    // Application specific
    Mover : REFERENCE TO FB_Mover;
END_VAR
VAR_OUTPUT
    (* standart Ausgänge *)
    xOUT_ErrFlag  : BOOL;            // Error Flag 
    xOUT_Busy     : BOOL;            // Baustein befindet sich im Ablauf 
    xOUT_Done     : BOOL;            // Baustein hat den Ablauf beendet 		
    xOUT_Ready    : BOOL;            // Ready to begin: should be the same state as done	
    xOUT_Timeout  : BOOL;            // Timeout FB 
    xOUT_InitDone : BOOL;            // initialisierung fertig
    xOUT_Wait     : BOOL;            // Wartet auf Bedingung
    iOUT_Step     : ST140_Measure_e; // Aktueller Schritt 
    sOUT_Step     : STRING;          // Aktueller Schritt but in string format
    bOUT_Error    : BYTE;            // Fehlernummer

    iOUT_ProcessCompletion : INT;  //process completion: express in % (0-100)
    xOUT_MoverFree         : BOOL; // The mover is free to move

END_VAR
VAR
    (* Standard *)
    (* Schritt *)
    iLastStep : ST140_Measure_e; // Merker letzter Schritt 
    iPreStep  : ST140_Measure_e; // Schritt zurück nach Alarm 
    iAktStep  : ST140_Measure_e; // aktueller Schritt

    // Trigger Starten 
    rtSTART : R_TRIG;
    // Timer TimeOut 
    TON_Timeout : TON;

    (* Bausteine *)
    arr_rMeasureTrack_Right : ARRAY[0..1] OF ARRAY[0..MEASURE_PER_PIECE - 1] OF REAL;
    arr_rMeasureTrack_Left  : ARRAY[0..1] OF ARRAY[0..MEASURE_PER_PIECE - 1] OF REAL;

    i            : INT;
    measureIndex : INT; // measure index

    testLevel_Min_Left_NOK  : BOOL; // TRUE when powder level is under the minimum
    testLevel_Max_Left_NOK  : BOOL; // TRUE when powder level is above the maximum
    testLevel_Min_Right_NOK : BOOL; // TRUE when powder level is under the minimum
    testLevel_Max_Right_NOK : BOOL; // TRUE when powder level is above the maximum

    visu_shuttle_x_position : LREAL; // position of the shuttle used in visu
	
	divisor_height_correction : LREAL := 4; // this divisor is used to reduce oscillation during height correction
	// because we may not fix the height on the very next shuttle

END_VAR
VAR CONSTANT
    MEASURE_SIMULATION : BOOL := FALSE; // Set to TRUE to simulate this part of the program
    MEASURE_PER_PIECE  : INT  := 3;     // this must be greater than 1 !
END_VAR

(*******************************************************************)
(* Trigger  *)
(*******************************************************************)
(* Zurücksetzen *)
IF xIN_RESET THEN
    iPreStep  := ST140_Measure_e.RESET;
    iOUT_Step := ST140_Measure_e.RESET;
END_IF;

(* Error Quittieren *)
IF (bOUT_Error <> 0) AND xIN_Quit THEN
    xOUT_ErrFlag := FALSE;
    bOUT_Error   := 0;
    iOUT_Step    := iPreStep; // iPreStep;
END_IF;

(*******************************************************************)
(* Timer *)
(*******************************************************************)
TON_Timeout(IN := xIN_NextStep AND (iLastStep = iOUT_Step) (*todo FG *) ,
            PT := tIN_Timeout);

(*******************************************************************)
(* Bausteine *)
(*******************************************************************)

(*******************************************************************)
(* OUTPUTS *)
(*******************************************************************)
// Error Flag
xOUT_ErrFlag := (bOUT_Error <> 0) OR (ST140_Measure_e.ERROR = iOUT_Step);
// Baustein befindet sich im Ablauf 
xOUT_Busy := (iOUT_Step > ST140_Measure_e.READY) AND (iOUT_Step < ST140_Measure_e.DONE);
// Baustein hat den Ablauf beendet
xOUT_Done := (iOUT_Step = ST140_Measure_e.DONE);
// Process ready
xOUT_Ready := (iOUT_Step = ST140_Measure_e.READY);
// Timeout FB 				 		
xOUT_Timeout := TON_Timeout.Q;
// Itialisierung fertig			
xOUT_InitDone := (iOUT_Step = ST140_Measure_e.READY) OR
                 (iOUT_Step = ST140_Measure_e.DONE);

// Aktueller Schritt			
iOUT_Step := iOUT_Step; //Im Ablauf gesetzt		
sOUT_Step := TO_STRING(iOUT_Step);
//Fehlernummer	 
bOUT_Error := bOUT_Error; //Im Ablauf/FB gesetzt	
(* Warte (alle Schritte wo auf FG oder Teile gewartet wird) *)
xOUT_Wait := (iOUT_Step = ST140_Measure_e.DONE) OR
             (iOUT_Step = ST140_Measure_e.READY) OR
             (iOUT_Step = ST140_Measure_e.START) OR
             (iOUT_Step = ST140_Measure_e.waitOnMover) OR
             (iOUT_Step = ST140_Measure_e.SYNC_MOVER_LEAVE);

xOUT_MoverFree :=
    NOT (iOUT_Step >= ST140_Measure_e.MOVER_NEEDED_OP AND iOUT_Step < ST140_Measure_e.MOVER_FREE_OP) AND
    (iOUT_Step >= ST140_Measure_e.READY) AND
    (iOUT_Step < ST140_Measure_e.ERROR);

iOUT_ProcessCompletion := F_GetPercent_2(iOUT_Step,
                                         ST140_Measure_e.waitOnMover,
                                         ST140_Measure_e.DONE,
                                         ST140_Measure_e.waitOnMover,
                                         ST140_Measure_e.DONE);

(*******************************************************************)
(* Ablauf *)
(*******************************************************************)

(* Sperren *)
IF xIN_Sperre THEN
    iPreStep  := ST140_Measure_e.RESET;
    iOUT_Step := ST140_Measure_e.RESET;
    RETURN;
END_IF;

(* Schritt Merker *)
IF iAktStep <> iOUT_Step THEN
    iLastStep := iAktStep;
    iAktStep  := iOUT_Step;
END_IF

(* START *)
rtSTART(CLK := xIN_Start);

IF __ISVALIDREF(Mover) THEN
    visu_shuttle_x_position := Mover.MovingProcessOffset;
ELSE
    visu_shuttle_x_position := 0.0;
END_IF

IF 0 = bOUT_Error THEN
    // put error conditions here
ELSIF iOUT_Step < ST140_Measure_e.ERROR THEN
    iOUT_Step := ST140_Measure_e.ERROR;
END_IF

(*******************************************************************)
(* Schrittkette  *)
(*******************************************************************)
CASE iOUT_Step OF

(***** RESET *****)
ST140_Measure_e.RESET: (* Schritt 0-99 *)
    //Initialisierungen
    //Start Init Ablauf
    IF xIN_Init THEN
        iOUT_Step := ST140_Measure_e.INIT;
        //Start Manu Ablauf
    ELSIF enIN_State = StateMANU AND xIN_NextStep THEN
        iOUT_Step := ST140_Measure_e.INIT;
    END_IF;

(***** INIT *****)
ST140_Measure_e.INIT: (* Grundstellung ? *)
    IF MEASURE_PER_PIECE < 2 THEN
        bOUT_Error := 4;
    END_IF

    iOUT_Step := ST140_Measure_e.READY;

(***** READY / INIT DONE *****)
ST140_Measure_e.READY: (* Start AUTO:END:LEER:STEP *)
    IF xIN_Start THEN  //IF rtSTART.Q THEN
        iOUT_Step := ST140_Measure_e.START;
    END_IF

(***** START  ZYKLISCH *****)
ST140_Measure_e.START: (*  *)
    IF xIN_NextStep AND pxFG_Freigabe^ THEN
        iOUT_Step := ST140_Measure_e.waitOnMover;
        iPreStep  := ST140_Measure_e.waitOnMover;
    END_IF;

ST140_Measure_e.waitOnMover:
    IF xIN_NextStep AND __ISVALIDREF(Mover) OR HMI.bArForceCyclusState[StationList_e.ST140] THEN
        IF Mover.GetLastStationDone() >= INT#140 THEN
            iOUT_Step := ST140_Measure_e.SYNC_MOVER_LEAVE;
        ELSIF Mover.GetLastStationDone() < INT#130 THEN
            iOUT_Step := ST140_Measure_e.SYNC_MOVER_LEAVE;
        ELSE
            MEMSET(ADR(arr_rMeasureTrack_Right), 0, SIZEOF(arr_rMeasureTrack_Right));
            MEMSET(ADR(arr_rMeasureTrack_Left), 0, SIZEOF(arr_rMeasureTrack_Left));

            measureIndex := 0;
            iOUT_Step    := ST140_Measure_e.Measure_right;
        END_IF
    END_IF

ST140_Measure_e.Measure_right:
    IF xIN_NextStep AND TRUE THEN
        arr_rMeasureTrack_Right[LaserPlace_e.NearTrack][measureIndex] :=
            UINT_TO_REAL(IN.AI01_ST140_level_track_side) * 0.001;

        arr_rMeasureTrack_Right[LaserPlace_e.NearDoor][measureIndex] :=
            UINT_TO_REAL(IN.AI02_ST140_level_door_side) * 0.001;

        measureIndex := measureIndex + 1;

        IF measureIndex >= MEASURE_PER_PIECE THEN
            IF _20_AUTO.recipe.st140.xIsTypeMiniOrSmart THEN
                iOUT_Step := ST140_Measure_e.Move_shuttle_to_pos_left;
            ELSE
                iOUT_Step := ST140_Measure_e.Save_result_in_mover;
            END_IF

            iOUT_Step := ST140_Measure_e.Move_shuttle_to_pos_left;
        ELSE
            iOUT_Step := ST140_Measure_e.Move_shuttle_relative_right;
        END_IF
    END_IF

ST140_Measure_e.Move_shuttle_relative_right:
    IF __ISVALIDREF(Mover) THEN
        IF Mover.MoveRelativeInsideStation(20.0 / (MEASURE_PER_PIECE - 1)) THEN
            iOUT_Step := ST140_Measure_e.Measure_right;
            iPreStep  := ST140_Measure_e.Measure_right;
        END_IF
    ELSE
        bOUT_Error := 10;
    END_IF

ST140_Measure_e.Move_shuttle_to_pos_left:
    IF __ISVALIDREF(Mover) THEN
        IF _20_AUTO.recipe.st140.xIsTypeMiniOrSmart THEN
            IF Mover.MoveRelativeInsideStation(100.0) THEN
                iOUT_Step    := ST140_Measure_e.Measure_left;
                iPreStep     := ST140_Measure_e.Measure_left;
                measureIndex := 0;
            END_IF
        ELSE
            iOUT_Step := ST140_Measure_e.Save_result_in_mover;
            iPreStep  := ST140_Measure_e.Save_result_in_mover;
        END_IF
    ELSE
        bOUT_Error := 11;
    END_IF

ST140_Measure_e.Measure_left:
    IF xIN_NextStep AND __ISVALIDREF(Mover) AND_THEN Mover.IsInStationPos() THEN
        arr_rMeasureTrack_Left[LaserPlace_e.NearTrack][measureIndex] :=
            UINT_TO_REAL(IN.AI01_ST140_level_track_side) * 0.001;

        arr_rMeasureTrack_Left[LaserPlace_e.NearDoor][measureIndex] :=
            UINT_TO_REAL(IN.AI02_ST140_level_door_side) * 0.001;

        measureIndex := measureIndex + 1;

        IF measureIndex >= MEASURE_PER_PIECE THEN
            iOUT_Step := ST140_Measure_e.Save_result_in_mover;
            iPreStep  := ST140_Measure_e.Save_result_in_mover;
        ELSE
            iOUT_Step := ST140_Measure_e.Move_shuttle_relative_left;
        END_IF
    END_IF

ST140_Measure_e.Move_shuttle_relative_left:
    IF __ISVALIDREF(Mover) THEN
        IF Mover.MoveRelativeInsideStation(20.0 / (MEASURE_PER_PIECE - 1)) THEN
            iOUT_Step := ST140_Measure_e.Measure_left;
            iPreStep  := ST140_Measure_e.Measure_left;
        END_IF
    ELSE
        bOUT_Error := 12;
    END_IF

ST140_Measure_e.Save_result_in_mover:

    testLevel_Min_Left_NOK  := FALSE;
    testLevel_Max_Left_NOK  := FALSE;
    testLevel_Min_Right_NOK := FALSE;
    testLevel_Max_Right_NOK := FALSE;

    IF NOT (MEASURE_SIMULATION AND CONST.USE_SIMULATION) THEN

        FOR i := 0 TO MEASURE_PER_PIECE - 1 BY 1 DO
            IF arr_rMeasureTrack_Right[LaserPlace_e.NearTrack][i] < _20_AUTO.recipe.st140.rMinHeightSensorRight OR
               arr_rMeasureTrack_Right[LaserPlace_e.NearDoor][i] < _20_AUTO.recipe.st140.rMinHeightSensorRight THEN
                // min value of the sensor means maximum fill
                testLevel_Max_Right_NOK := TRUE;
            END_IF

            IF arr_rMeasureTrack_Right[LaserPlace_e.NearTrack][i] > _20_AUTO.recipe.st140.rMaxHeightSensorRight OR
               arr_rMeasureTrack_Right[LaserPlace_e.NearDoor][i] > _20_AUTO.recipe.st140.rMaxHeightSensorRight THEN
                // max value of the sensor means minimum fill
                testLevel_Min_Right_NOK := TRUE;
            END_IF
        END_FOR

        IF _20_AUTO.recipe.st140.xIsTypeMiniOrSmart THEN
            FOR i := 0 TO MEASURE_PER_PIECE - 1 BY 1 DO
                IF arr_rMeasureTrack_Left[LaserPlace_e.NearTrack][i] < _20_AUTO.recipe.st140.rMinHeightSensorLeft OR
                   arr_rMeasureTrack_Left[LaserPlace_e.NearDoor][i] < _20_AUTO.recipe.st140.rMinHeightSensorLeft THEN
                    // min value of the sensor means maximum fill
                    testLevel_Max_Left_NOK := TRUE;
                END_IF

                IF arr_rMeasureTrack_Left[LaserPlace_e.NearTrack][i] > _20_AUTO.recipe.st140.rMaxHeightSensorLeft OR
                   arr_rMeasureTrack_Left[LaserPlace_e.NearDoor][i] > _20_AUTO.recipe.st140.rMaxHeightSensorLeft THEN
                    // max value of the sensor means minimum fill
                    testLevel_Min_Left_NOK := TRUE;
                END_IF
            END_FOR
        END_IF

    END_IF

    IF testLevel_Min_Left_NOK OR testLevel_Max_Left_NOK OR testLevel_Min_Right_NOK OR testLevel_Max_Right_NOK THEN
        IF __ISVALIDREF(Mover) THEN
            IF NOT Mover.SetLastStation(-140) THEN
                ASSERT(0);
            END_IF

            // All minimum
            IF (testLevel_Min_Left_NOK AND testLevel_Min_Right_NOK) THEN
                Mover.SetErrorCode(CONCAT(INT_TO_STRING(Mover.GetLastStationDone()), '-D All min'));

                // All maximum
            ELSIF (testLevel_Max_Left_NOK AND testLevel_Max_Right_NOK) THEN
                Mover.SetErrorCode(CONCAT(INT_TO_STRING(Mover.GetLastStationDone()), '-E All max'));

                // Both in error
            ELSIF (testLevel_Min_Left_NOK OR testLevel_Max_Left_NOK) AND
                  (testLevel_Min_Right_NOK OR testLevel_Max_Right_NOK) THEN
                Mover.SetErrorCode(CONCAT(INT_TO_STRING(Mover.GetLastStationDone()), '-F Both left and right'));

                // min and max error on left
            ELSIF (testLevel_Min_Left_NOK AND testLevel_Max_Left_NOK) THEN
                Mover.SetErrorCode(CONCAT(INT_TO_STRING(Mover.GetLastStationDone()), '-G Both left'));

                // min and max error on right
            ELSIF (testLevel_Min_Right_NOK AND testLevel_Max_Right_NOK) THEN
                Mover.SetErrorCode(CONCAT(INT_TO_STRING(Mover.GetLastStationDone()), '-H Both right'));

            ELSIF testLevel_Min_Left_NOK THEN
                Mover.SetErrorCode(CONCAT(INT_TO_STRING(Mover.GetLastStationDone()), '-I Min left'));

            ELSIF testLevel_Max_Left_NOK THEN
                Mover.SetErrorCode(CONCAT(INT_TO_STRING(Mover.GetLastStationDone()), '-J Max left'));

            ELSIF testLevel_Min_Right_NOK THEN
                Mover.SetErrorCode(CONCAT(INT_TO_STRING(Mover.GetLastStationDone()), '-K Min right'));

            ELSIF testLevel_Max_Right_NOK THEN
                Mover.SetErrorCode(CONCAT(INT_TO_STRING(Mover.GetLastStationDone()), '-L Min right'));

            ELSE
                ASSERT(0); // Oops ... read the condition again !
            END_IF
        END_IF

    ELSE
        IF __ISVALIDREF(Mover) THEN
            IF NOT Mover.SetLastStation(140) THEN
                ASSERT(0);
            END_IF
        END_IF
    END_IF

	// Adding a value makes the axis go down
	// Substracting a value makes the axis go up
    IF __ISVALIDREF(Mover) AND_THEN Mover.GetLastStationDone() = 130 THEN
        IF testLevel_Min_Left_NOK THEN
            GVL.ST130_01Y_Feedback_Offset := GVL.ST130_01Y_Feedback_Offset - 0.1;
        END_IF
        IF testLevel_Max_Left_NOK THEN
            GVL.ST130_01Y_Feedback_Offset := GVL.ST130_01Y_Feedback_Offset + 0.1;
        END_IF
        IF testLevel_Min_Right_NOK THEN
            GVL.ST130_01Y_Feedback_Offset := GVL.ST130_01Y_Feedback_Offset - 0.1;
        END_IF
        IF testLevel_Max_Right_NOK THEN
            GVL.ST130_01Y_Feedback_Offset := GVL.ST130_01Y_Feedback_Offset + 0.1;
        END_IF
    END_IF

	// Adding a value makes the axis go down
	// Substracting a value makes the axis go up
    IF __ISVALIDREF(Mover) AND_THEN Mover.GetLastStationDone() = 135 THEN
        IF testLevel_Min_Left_NOK THEN
            GVL.ST135_01Y_Feedback_Offset := GVL.ST135_01Y_Feedback_Offset - 0.1;
        END_IF
        IF testLevel_Max_Left_NOK THEN
            GVL.ST135_01Y_Feedback_Offset := GVL.ST135_01Y_Feedback_Offset + 0.1;
        END_IF
        IF testLevel_Min_Right_NOK THEN
            GVL.ST135_01Y_Feedback_Offset := GVL.ST135_01Y_Feedback_Offset - 0.1;
        END_IF
        IF testLevel_Max_Right_NOK THEN
            GVL.ST135_01Y_Feedback_Offset := GVL.ST135_01Y_Feedback_Offset + 0.1;
        END_IF
    END_IF

    iOUT_Step := ST140_Measure_e.SYNC_MOVER_LEAVE;

ST140_Measure_e.SYNC_MOVER_LEAVE:
    // The mover needs to be taken by MoverMan
    IF NOT __ISVALIDREF(Mover) THEN
        iOUT_Step := ST140_Measure_e.DONE;
    END_IF

(***** DONE *****)
ST140_Measure_e.DONE: (* Letzter Schritt  *)
    IF NOT xIN_AlarmAktiv THEN
        //AUTO
        IF (enIN_State = StateAUTO) AND xIN_RestartCYCL THEN
            iOUT_Step := ST140_Measure_e.START;
            //STEP / END / LEERFAHREN restart
        ELSIF (enIN_State < StateAUTO) AND (enIN_State >= enState.StateSTEP) AND xIN_RestartCYCL THEN
            iOUT_Step := ST140_Measure_e.START;
            //STEP / END / LEERFAHREN fertig
        ELSIF (enIN_State = StateREADY) THEN
            iOUT_Step := ST140_Measure_e.READY;
        END_IF;
    END_IF;

(************ ERROR *************)
ST140_Measure_e.ERROR: (* ERROR *) ;

END_CASE;

END_FUNCTION_BLOCK

// ---- POUs/20_AUTO/ST145/FB_AUT_145.TcPOU
FUNCTION_BLOCK FB_AUT_145 EXTENDS FB_AUT_ABSTRACT
(****************************************************************************)
(*	POU_AUT_zxx			Bausteinaufrufe Station	zxx							*)
(*	Status				ungetestet											*)
(*  Version:			1.0													*)
(*	Beschrieb:																*)
(*																			*)
(*	Abläufe:			FB_ABLzxxA		Hauptablauf							*)
(*																			*)
(*																			*)
(* 	25.09.2019/Dj															*)
(****************************************************************************)
(*	dd.mm.yyyy   KZ    x.y			Beschrieb								*)
(****************************************************************************)
VAR_INPUT
    (* spezifische Eingänge *)

END_VAR
VAR_OUTPUT
    (* spezifische Ausgänge *)

END_VAR
VAR
    (* Bausteine *)
    fb_Pnp    : FB_ABL_145_Pnp;
    fb_Feeder : FB_ABL_145_Feeder;

    fb_stat_pnp    : FB_AUT_Statistics;
    fb_stat_Feeder : FB_AUT_Statistics;

END_VAR

VAR CONSTANT
    ROT_TABLE_FREE_MAX_Y : REAL := 200.0; // If Y and Z axis is more than this value, the feeder cannot move
    ROT_TABLE_FREE_MAX_Z : REAL := 200.0; // If Z and Y axis is more than this value, the feeder cannot move

    PNP_VERTICAL_MAX_Z : REAL := 50.0; // If Z axis is more than this value, the horizontal axis of the pnp cannot move
END_VAR

(*******************************************************************)
(* Timer *)
(*******************************************************************)

(*******************************************************************)
(* Flanken / Merker *)
(*******************************************************************)
//MANU CYCLE
IF (enIN_State = StateMANU) AND xIN_ManuCycle THEN
    xManuCycle := TRUE;
END_IF;

IF (enIN_State <> StateMANU) OR xOUT_Done THEN
    xManuCycle := FALSE;
END_IF

//NEXT STEP
xNextStep := (enIN_State > StateSTEP) OR
             ((enIN_State = StateSTEP) AND xIN_Step) OR
             ((enIN_State = StateMANU) AND xManuCycle);

//RESET
xReset := (enIN_State < StateREADY) AND (enIN_State <> StateINIT) AND NOT xManuCycle;

(*******************************************************************)
(* Bausteinaufrufe Abläufe *)
(*******************************************************************)

xRelease := MAIN.MoverMan.IsProcessUsed(THIS^);

fb_Pnp(xIN_Reset          := xReset,
       xIN_Init           := xIN_Init,
       xIN_Quit           := xIN_Quit,
       xIN_Start          := enIN_State >= enState.StateLEER AND xRelease,
       xIN_Sperre         := NOT xIN_On,
       xIN_NextStep       := xNextStep,
       xIN_AlarmAktiv     := xIN_AlarmAktiv,
       xIN_DryCycle       := xIN_DryCycle,
       xIN_RestartCYCL    := enIN_State >= enState.StateLEER,
       enIN_State         := enIN_State,
       tIN_Timeout        := tIN_Timeout,
       pxFG_Freigabe      := ADR(xRelease),
       Mover              := THIS^.Mover,
       xIN_PceReadyToPick := fb_Feeder.xOUT_Done,
       xIN_HorAxisFree    := ST145_Axis.axis145_02Z.rActPos < ROT_TABLE_FREE_MAX_Y);

fb_Feeder(xIN_Reset       := xReset,
          xIN_Init        := xIN_Init,
          xIN_Quit        := xIN_Quit,
          xIN_Start       := enIN_State >= enState.StateLEER AND xRelease,
          xIN_Sperre      := NOT xIN_On,
          xIN_NextStep    := xNextStep,
          xIN_AlarmAktiv  := xIN_AlarmAktiv,
          xIN_DryCycle    := xIN_DryCycle,
          xIN_RestartCYCL := enIN_State >= enState.StateLEER,
          enIN_State      := enIN_State,
          tIN_Timeout     := tIN_Timeout,
          pxFG_Freigabe   := ADR(xRelease),
          // special
          xIN_PickPiece            := fb_Pnp.xOUT_PickPiece,
          xIN_RotTableBlockedByPnp := (ST145_Axis.axis145_01Y.rActPos > ROT_TABLE_FREE_MAX_Y) AND
                                      (ST145_Axis.axis145_02Z.rActPos > ROT_TABLE_FREE_MAX_Z));

fb_stat_pnp(xIN_Enable  := enState.StateAUTO = enIN_State,
            xIN_Waiting := fb_Pnp.xOUT_Wait,
            xIN_Running := (fb_Pnp.iOUT_Step >= ST145_Pnp_e.START) AND
                           (fb_Pnp.iOUT_Step <= ST145_Pnp_e.DONE),
            // Since we use a mover system, a cycle is done when we are waiting on a mover
            xIN_Done := fb_Pnp.iOUT_Step = ST145_Pnp_e.waitOnMover);

fb_stat_Feeder(xIN_Enable  := enState.StateAUTO = enIN_State,
               xIN_Waiting := fb_feeder.xOUT_Wait,
               xIN_Running := (fb_feeder.iOUT_Step >= ST145_Feeder_e.START) AND
                              (fb_feeder.iOUT_Step <= ST145_Feeder_e.DONE),
               xIN_Done := fb_feeder.iOUT_Step = ST145_Feeder_e.DONE);

(*******************************************************************)
(* Mover reset flags *)
(*******************************************************************)

(*******************************************************************)
(* OUTPUT *)
(*******************************************************************)
xOUT_InitDone := fb_Pnp.xOUT_InitDone AND fb_Feeder.xOUT_InitDone;
xOUT_Ready    := fb_Pnp.xOUT_Ready AND fb_Feeder.xOUT_Ready;
xOUT_Done     := fb_Pnp.xOUT_Done; // we ignore feeder
xOUT_ErrFlag  := fb_Pnp.xOUT_ErrFlag OR fb_Feeder.xOUT_ErrFlag;
xOUT_Wait     := fb_Pnp.xOUT_Wait AND fb_Feeder.xOUT_Wait;
xOUT_AlarmST  := xOUT_ErrFlag;

(*******************************************************************)
(* Bausteinaufruf Error Station *)
(*******************************************************************)
// POU_ERR_VORLAGE(xIN_QUIT:=xIN_Quit , pstrArIN_ALARM:=ADR(HMI.strArALARM[1]));

(* % of completion of the process *)
PROPERTY iCompletionPC : INT
GET
iCompletionPC := THIS^.fb_Pnp.iOUT_ProcessCompletion;
END_GET
END_PROPERTY

PROPERTY ProcessExecution : ProcessExecution_e
GET
ProcessExecution := THIS^._ProcessExecution;
END_GET
SET
THIS^._ProcessExecution := ProcessExecution;
END_SET
END_PROPERTY

PROPERTY xBusy : BOOL
GET
xBusy := THIS^.fb_Pnp.xOUT_Busy;
END_GET
SET
END_SET
END_PROPERTY

PROPERTY xDone : BOOL
GET
xDone := THIS^.fb_Pnp.xOUT_Ready OR THIS^.fb_Pnp.xOUT_Done;
END_GET
END_PROPERTY

PROPERTY xMoverPathFree : BOOL
GET
xMoverPathFree := THIS^.fb_Pnp.xOUT_MoverFree OR THIS^.fb_Pnp.xOUT_Ready OR THIS^.fb_Pnp.xOUT_Done;
END_GET
END_PROPERTY

PROPERTY xMoverShouldLeave : BOOL
GET
xMoverShouldLeave := THIS^.fb_Pnp.iOUT_Step = ST145_Pnp_e.SYNC_MOVER_LEAVE;
END_GET
END_PROPERTY

END_FUNCTION_BLOCK

// ---- POUs/20_AUTO/ST145/FB_ABL_145_Pnp.TcPOU
FUNCTION_BLOCK FB_ABL_145_Pnp
(****************************************************************************************)
(*	TITEL				laden kristall- Modul	    										*)
(*	Status				ungetestet                         								*)
(*	Beschrieb:			Ablaufbeschreibung												*)
(*																						*)
(*	Steps:	self-explained using enum													*)
(***********************************Revisionen*******************************************)
(*	see github blames																	*)
(****************************************************************************************)

VAR_INPUT
    xIN_Reset       : BOOL;          // Schrittkette zurücksetzen 
    xIN_Init        : BOOL;          // Initialisieren
    xIN_Quit        : BOOL;          // Fehler quittieren 
    xIN_Start       : BOOL;          // Startbefehl
    xIN_Sperre      : BOOL;          // FB Sperren 
    xIN_NextStep    : BOOL;          // Nächsten Schritt ausführen 
    xIN_AlarmAktiv  : BOOL;          // Anlage hat Alarm
    xIN_DryCycle    : BOOL;          // Fahren ohne Teile
    xIN_RestartCYCL : BOOL;          // Zyklus erneut starten im STEP, END, LEERFAHREN
    enIN_State      : enState;       // Status Anlage
    tIN_Timeout     : TIME := T#10s; // Timout

    pxFG_Freigabe : POINTER TO BOOL; //Freigabe von Station

    // Application specific
    Mover              : REFERENCE TO FB_Mover;
    xIN_PceReadyToPick : BOOL; // the piece(s) is/are ready to picked
    xIN_HorAxisFree    : BOOL; // TRUE when the vertical is up enough
END_VAR
VAR_OUTPUT
    (* standart Ausgänge *)
    xOUT_ErrFlag  : BOOL;        // Error Flag 
    xOUT_Busy     : BOOL;        // Baustein befindet sich im Ablauf 
    xOUT_Done     : BOOL;        // Baustein hat den Ablauf beendet 		
    xOUT_Ready    : BOOL;        // Ready to begin, should be the same state as done	
    xOUT_Timeout  : BOOL;        // Timeout FB 
    xOUT_InitDone : BOOL;        // initialisierung fertig
    xOUT_Wait     : BOOL;        // Wartet auf Bedingung
    iOUT_Step     : ST145_Pnp_e; // Aktueller Schritt 
    sOUT_Step     : STRING;      // Aktueller Schritt but in string format
    bOUT_Error    : BYTE;        // Fehlernummer

    iOUT_ProcessCompletion : INT;  //process completion, express in % (0-100)
    xOUT_MoverFree         : BOOL; // The mover is free to move
    xOUT_PickPiece         : BOOL; // Set to true when a piece is picked

END_VAR
VAR
    (* Standard *)
    (* Schritt *)
    iLastStep : ST145_Pnp_e; // Merker letzter Schritt 
    iPreStep  : ST145_Pnp_e; // Schritt zurück nach Alarm 
    iAktStep  : ST145_Pnp_e; // aktueller Schritt

    // Trigger Starten 
    rtSTART : R_TRIG;
    // Timer TimeOut 
    TON_Timeout : TON;

    (* Bausteine *)

    (* Spezial *)
    fb_axis145_01Y : FB_AxisLM_V1_1;
    fb_axis145_02Z : FB_AxisLM_V1_1;

    fb_PnpHorAxis : FB_LinearMotionMan;
    fb_PnpVerAxis : FB_LinearMotionMan;

    fb_simu_axis145_01Y : FB_Simu_AxisLM_V1_1;
    fb_simu_axis145_02Z : FB_Simu_AxisLM_V1_1;

    fb_vakumGriperLeft    : FB_ZylMo2El_V2_1;
    fb_vakumGriperRight   : FB_ZylMo2El_V2_1;
    simu_vacumGriperLeft  : FB_Simu_Zyl2Pos;
    simu_vacumGriperRight : FB_Simu_Zyl2Pos;

END_VAR
VAR CONSTANT
    PNP_SIMULATION : BOOL := FALSE; // Set to TRUE to simulate this part of the program
END_VAR

(*******************************************************************)
(* Trigger  *)
(*******************************************************************)
(* Zurücksetzen *)
IF xIN_RESET THEN
    iPreStep  := ST145_Pnp_e.RESET;
    iOUT_Step := ST145_Pnp_e.RESET;
END_IF;

(* Error Quittieren *)
IF (bOUT_Error <> 0) AND xIN_Quit THEN
    xOUT_ErrFlag := FALSE;
    bOUT_Error   := 0;
    iOUT_Step    := iPreStep;
END_IF;

(*******************************************************************)
(* Timer *)
(*******************************************************************)
TON_Timeout(IN := xIN_NextStep AND (iLastStep = iOUT_Step) (*todo FG *) ,
            PT := tIN_Timeout);

(*******************************************************************)
(* Bausteine *)
(*******************************************************************)
fb_PnpHorAxis(config          := _20_AUTO.recipe.linearAxis[LinearAxis_e.ST145_01Y],
              xIN_Init        := enIN_State = enState.StateINIT,
              xIN_Reset       := xIN_Reset,
              lrIN_CurrPos    := fb_axis145_01Y.rOUT_ActPos,
              lrIN_Delta_mm   := 0.5,
              iIN_CurrentStep := iOUT_Step,
              iIN_moveNumber  := ST145_PnpHorPos_e._max);

fb_simu_axis145_01Y(xIN_Enable          := PNP_SIMULATION AND CONST.USE_SIMULATION,
                    bIN_AxisCntr        := fb_axis145_01Y.bOUT_AxisCntr,
                    wIN_AxisState       := ST145_Axis.axis145_01Y.wState,
                    udiIN_HomingTime_ms := 2000,
                    pIN_axisSimu        := ADR(SIMU.axis_ref[Axis_e.ST145_01Y]),
                    pIN_axisHW          := ADR(ST145_Axis.axis145_01Y.axis),
                    rIN_PosActual       := fb_axis145_01Y.rOUT_ActPos,
                    rIN_PosMax          := ST145_Axis.const145_01Y.POS_MAX,
                    rIN_PosMin          := ST145_Axis.const145_01Y.POS_MIN,
                    rIN_PixMax          := 100,
                    rIN_PixMin          := 0);

fb_axis145_01Y(enIN_State       := enIN_State,
               parIN_Buttons    := ADR(AXIS.btTeachArAxis[Axis_e.ST145_01Y]),
               xIN_DisButtons   :=,
               xIN_Quit         := xIN_Quit,
               xIN_PARAMok      := TRUE, (*TODO*)
               xIN_FREE         := TRUE,
               xIN_FREE_HOME    := TRUE,
               rIN_POSMIN       := ST145_Axis.const145_01Y.POS_MIN,
               rIN_POSMAX       := ST145_Axis.const145_01Y.POS_MAX,
               rIN_VELOMAX      := ST145_Axis.const145_01Y.VELO_MAX,
               rIN_VELOMANU     := ST145_Axis.const145_01Y.VELO_MANU,
               rIN_VELOOPEN     := ST145_Axis.const145_01Y.VELO_MANU / 4,
               rIN_JogInc       := AXIS.rTeachIncAxis,
               xIN_Execute      := fb_PnpHorAxis.xOUT_Execute,
               xIN_Home         := ST145_Pnp_e.Init_HomeHorizontals = iAktStep,
               xIN_Relative     :=,
               rIN_Position     := TO_REAL(fb_PnpHorAxis.OUT_MoveProfile.lrPosition),
               rIN_Velocity     := TO_REAL(fb_PnpHorAxis.OUT_MoveProfile.lrVelocity),
               rIN_Acceleration := TO_REAL(fb_PnpHorAxis.OUT_MoveProfile.lrAccel),
               rIN_Deceleration := TO_REAL(fb_PnpHorAxis.OUT_MoveProfile.lrDecel),
               rIN_Jerk         := TO_REAL(fb_PnpHorAxis.OUT_MoveProfile.lrJerk),
               rIN_PosManu      :=
               TO_REAL(_20_AUTO.recipe
                           .linearAxis[LinearAxis_e.ST145_01Y].movesList[AXIS.bTeachPos[Axis_e.ST145_01Y]].lrPosition),
               rIN_VeloJogManu := TO_REAL(Axis.rJogVelo_pc),
               xIN_Reset       := (ST145_Pnp_e.RESET = iAktStep) OR xIN_Reset,
               // The simu fb gives the hardware state when we are not in simu
               wAxisState    := fb_simu_axis145_01Y.wOUT_AxisState,
               rOUT_ActPos   => st145_axis.axis145_01Y.rActPos,
               bOUT_AxisCntr => ST145_Axis.axis145_01Y.bCtrlHi,
               axisIN_REF    := fb_simu_axis145_01Y.pOUT_axisRef^);

fb_PnpVerAxis(config          := _20_AUTO.recipe.linearAxis[LinearAxis_e.ST145_02Z],
              xIN_Init        := enIN_State = enState.StateINIT,
              xIN_Reset       := xIN_Reset,
              lrIN_CurrPos    := fb_axis145_02Z.rOUT_ActPos,
              lrIN_Delta_mm   := 1.0,
              iIN_CurrentStep := iOUT_Step,
              iIN_moveNumber  := ST145_PnpVerPos_e._max);

fb_simu_axis145_02Z(xIN_Enable          := PNP_SIMULATION AND CONST.USE_SIMULATION,
                    bIN_AxisCntr        := fb_axis145_02Z.bOUT_AxisCntr,
                    wIN_AxisState       := ST145_Axis.axis145_02Z.wState,
                    udiIN_HomingTime_ms := 2000,
                    pIN_axisSimu        := ADR(SIMU.axis_ref[Axis_e.ST145_02Z]),
                    pIN_axisHW          := ADR(ST145_Axis.axis145_02Z.axis),
                    rIN_PosActual       := fb_axis145_02Z.rOUT_ActPos,
                    rIN_PosMax          := ST145_Axis.const145_02Z.POS_MAX,
                    rIN_PosMin          := ST145_Axis.const145_02Z.POS_MIN,
                    rIN_PixMax          := 100,
                    rIN_PixMin          := 0);

fb_axis145_02Z(enIN_State       := enIN_State,
               parIN_Buttons    := ADR(AXIS.btTeachArAxis[Axis_e.ST145_02Z]),
               xIN_DisButtons   :=,
               xIN_Quit         := xIN_Quit,
               xIN_PARAMok      := TRUE, (*TODO*)
               xIN_FREE         := TRUE,
               xIN_FREE_HOME    := TRUE,
               rIN_POSMIN       := ST145_Axis.const145_02Z.POS_MIN,
               rIN_POSMAX       := ST145_Axis.const145_02Z.POS_MAX,
               rIN_VELOMAX      := ST145_Axis.const145_02Z.VELO_MAX,
               rIN_VELOMANU     := ST145_Axis.const145_02Z.VELO_MANU,
               rIN_VELOOPEN     := ST145_Axis.const145_02Z.VELO_MANU / 4,
               rIN_JogInc       := AXIS.rTeachIncAxis,
               xIN_Execute      := fb_PnpVerAxis.xOUT_Execute,
               xIN_Home         := ST145_Pnp_e.Init_HomeVerticals = iAktStep,
               xIN_Relative     :=,
               rIN_Position     := TO_REAL(fb_PnpVerAxis.OUT_MoveProfile.lrPosition),
               rIN_Velocity     := TO_REAL(fb_PnpVerAxis.OUT_MoveProfile.lrVelocity),
               rIN_Acceleration := TO_REAL(fb_PnpVerAxis.OUT_MoveProfile.lrAccel),
               rIN_Deceleration := TO_REAL(fb_PnpVerAxis.OUT_MoveProfile.lrDecel),
               rIN_Jerk         := TO_REAL(fb_PnpVerAxis.OUT_MoveProfile.lrJerk),
               rIN_PosManu      :=
               TO_REAL(_20_AUTO.recipe
                           .linearAxis[LinearAxis_e.ST145_02Z].movesList[AXIS.bTeachPos[Axis_e.ST145_02Z]].lrPosition),
               rIN_VeloJogManu := TO_REAL(Axis.rJogVelo_pc),
               xIN_Reset       := (ST145_Pnp_e.RESET = iAktStep) OR xIN_Reset,
               // The simu fb gives the hardware state when we are not in simu
               wAxisState    := fb_simu_axis145_02Z.wOUT_AxisState,
               rOUT_ActPos   => st145_axis.axis145_02Z.rActPos,
               bOUT_AxisCntr => ST145_Axis.axis145_02Z.bCtrlHi,
               axisIN_REF    := fb_simu_axis145_02Z.pOUT_axisRef^);

//////////////////////////////////
fb_vakumGriperLeft(xIN_Reset    := xIN_Reset OR (ST145_Pnp_e.RESET = iOUT_Step),
                   xIN_Quit     := xIN_Quit,
                   xIN_Manu     := enState.StateMANU = enIN_State,
                   pbtIN_Button := ADR(HMI.btManuCylinders[StationList_e.ST145][1]),
                   xIN_GS       := simu_vacumGriperLeft.xOUT_inGS,
                   xIN_AS       := simu_vacumGriperLeft.xOUT_inAS,
                   xIN_FREE     := TRUE,
                   xINtoGS      := ST145_Pnp_e.Vacum_off = iOUT_Step,
                   xINtoAS      := _20_AUTO.recipe.st145.xUseVerLeft AND ST145_Pnp_e.Vacum_on = iOUT_Step,
                   tIN_ErrAS    := DINT_TO_TIME(_20_AUTO.recipe.cylinder2Pos[StationList_e.ST145]
                                                    [ST145_Cylinders_e.VakuumgreiferLinks].toAS_alarm_time),
                   tIN_ErrGS := DINT_TO_TIME(_20_AUTO.recipe.cylinder2Pos[StationList_e.ST145]
                                                 [ST145_Cylinders_e.VakuumgreiferLinks].toGS_alarm_time),
                   tIN_WaitAS := DINT_TO_TIME(_20_AUTO.recipe.cylinder2Pos[StationList_e.ST145]
                                                  [ST145_Cylinders_e.VakuumgreiferLinks].toAS_wait_time),
                   tIN_WaitGS := DINT_TO_TIME(_20_AUTO.recipe.cylinder2Pos[StationList_e.ST145]
                                                  [ST145_Cylinders_e.VakuumgreiferLinks].toGS_wait_time));

simu_vacumGriperLeft(xIN_Enable := PNP_SIMULATION AND CONST.USE_SIMULATION,
                     xIN_inGS   := NOT IO_BOX.I1600_ST145_vakum_teil_in_greiffer_left,
                     xIN_inAS   := IO_BOX.I1600_ST145_vakum_teil_in_greiffer_left,
                     xIN_valve  := fb_vakumGriperLeft.xOUT_VALVE,
                     tIN_GS_ms  := 0,    //ms
                     tIN_AS_ms  := 200); //ms

fb_vakumGriperRight(xIN_Reset    := xIN_Reset OR (ST145_Pnp_e.RESET = iOUT_Step),
                    xIN_Quit     := xIN_Quit,
                    xIN_Manu     := enState.StateMANU = enIN_State,
                    pbtIN_Button := ADR(HMI.btManuCylinders[StationList_e.ST145][2]),
                    xIN_GS       := simu_vacumGriperRight.xOUT_inGS,
                    xIN_AS       := simu_vacumGriperRight.xOUT_inAS,
                    xIN_FREE     := TRUE,
                    xINtoGS      := ST145_Pnp_e.Vacum_off = iOUT_Step,
                    xINtoAS      := _20_AUTO.recipe.st145.xUseVerRight AND ST145_Pnp_e.Vacum_on = iOUT_Step,
                    tIN_ErrAS    := DINT_TO_TIME(_20_AUTO.recipe.cylinder2Pos[StationList_e.ST145]
                                                     [ST145_Cylinders_e.VakuumgreiferRechts].toAS_alarm_time),
                    tIN_ErrGS := DINT_TO_TIME(_20_AUTO.recipe.cylinder2Pos[StationList_e.ST145]
                                                  [ST145_Cylinders_e.VakuumgreiferRechts].toGS_alarm_time),
                    tIN_WaitAS := DINT_TO_TIME(_20_AUTO.recipe.cylinder2Pos[StationList_e.ST145]
                                                   [ST145_Cylinders_e.VakuumgreiferRechts].toAS_wait_time),
                    tIN_WaitGS := DINT_TO_TIME(_20_AUTO.recipe.cylinder2Pos[StationList_e.ST145]
                                                   [ST145_Cylinders_e.VakuumgreiferRechts].toGS_wait_time));

simu_vacumGriperRight(xIN_Enable := PNP_SIMULATION AND CONST.USE_SIMULATION,
                      xIN_inGS   := NOT IO_BOX.I1601_ST145_vakum_teil_in_greiffer_right,
                      xIN_inAS   := IO_BOX.I1601_ST145_vakum_teil_in_greiffer_right,
                      xIN_valve  := fb_vakumGriperRight.xOUT_VALVE,
                      tIN_GS_ms  := 0,    //ms
                      tIN_AS_ms  := 200); //ms

(*******************************************************************)
(* OUTPUTS *)
(*******************************************************************)
// Error Flag 
xOUT_ErrFlag := (bOUT_Error <> 0) OR (ST145_Pnp_e.ERROR = iOUT_Step);
// Baustein befindet sich im Ablauf 
xOUT_Busy := (iOUT_Step > ST145_Pnp_e.READY) AND (iOUT_Step < ST145_Pnp_e.DONE);
// Baustein hat den Ablauf beendet
xOUT_Done := (iOUT_Step = ST145_Pnp_e.DONE);
// Process ready
xOUT_Ready := (iOUT_Step = ST145_Pnp_e.READY) OR (iOUT_Step = ST145_Pnp_e.waitOnMover);
// Timeout FB 				 		
xOUT_Timeout := TON_Timeout.Q;
// Itialisierung fertig			
xOUT_InitDone := (iOUT_Step = ST145_Pnp_e.READY) OR (iOUT_Step = ST145_Pnp_e.waitOnMover);
// Aktueller Schritt			
iOUT_Step := iOUT_Step; //Im Ablauf gesetzt		
sOUT_Step := TO_STRING(iOUT_Step);
//Fehlernummer	 
bOUT_Error := bOUT_Error; //Im Ablauf/FB gesetzt	
(* Warte (alle Schritte wo auf FG oder Teile gewartet wird) *)
xOUT_Wait := (iOUT_Step = ST145_Pnp_e.DONE) OR
             (iOUT_Step = ST145_Pnp_e.READY) OR
             (iOUT_Step = ST145_Pnp_e.START) OR
             (iOUT_Step = ST145_Pnp_e.waitOnMover) OR
             (iOUT_Step = ST145_Pnp_e.SYNC_MOVER_LEAVE) OR
             (iOUT_Step = ST145_Pnp_e.PnP_WaitOnFeeder);

xOUT_MoverFree := iOUT_Step >= ST145_Pnp_e.MOVER_FREE_OP AND iOUT_Step < ST145_Pnp_e.MOVER_NEEDED_OP;

iOUT_ProcessCompletion := F_GetPercent_2(iAktStep,
                                         ST145_Pnp_e.Pnp_Hor_ToRotTablePos,
                                         ST145_Pnp_e.Pnp_Hor_ToTrackPos,
                                         ST145_Pnp_e.Pnp_Ver_ShuttleDown,
                                         ST145_Pnp_e.SYNC_MOVER_LEAVE);

xOUT_PickPiece := iOUT_Step = ST145_Pnp_e.Vacum_on; // the feeder needs to move only when 
// the pnp is outside the feeder

// TODO Valve should not be set when we are in simulation !
IO_BOX.Q0200_14_ST145_vakum_greifer_links :=
    fb_vakumGriperLeft.xOUT_VALVE AND NOT (PNP_SIMULATION AND CONST.USE_SIMULATION);

IO_BOX.Q0201_14_ST145_vakum_greifer_rechts :=
    fb_vakumGriperRight.xOUT_VALVE AND NOT (PNP_SIMULATION AND CONST.USE_SIMULATION);

(*******************************************************************)
(* Ablauf *)
(*******************************************************************)

(* Sperren *)
IF xIN_Sperre THEN
    iPreStep  := ST145_Pnp_e.RESET;
    iOUT_Step := ST145_Pnp_e.RESET;
    RETURN;
END_IF;

(* Schritt Merker *)
IF iAktStep <> iOUT_Step THEN
    iLastStep := iAktStep;
    iAktStep  := iOUT_Step;
END_IF

(* START *)
rtSTART(CLK := xIN_Start);

IF 0 = bOUT_Error THEN
    IF fb_axis145_01Y.xOUT_ErrFlag THEN
        bOUT_Error := 11;
    ELSIF fb_axis145_02Z.xOUT_ErrFlag THEN
        bOUT_Error := 12;
    ELSIF fb_vakumGriperLeft.xOUT_ErrFlag THEN
        bOUT_Error := 13;
    ELSIF fb_vakumGriperRight.xOUT_ErrFlag THEN
        bOUT_Error := 14;
    END_IF
ELSIF iOUT_Step < ST145_Pnp_e.ERROR THEN
    iPreStep  := ST145_Pnp_e.INIT;
    iOUT_Step := ST145_Pnp_e.ERROR;
END_IF

(*******************************************************************)
(* Schrittkette  *)
(*******************************************************************)
CASE iOUT_Step OF

(***** RESET *****)
ST145_Pnp_e.RESET: (* Schritt 0-99 *)
    //Initialisierungen
    //Start Init Ablauf
    IF xIN_Init THEN
        iOUT_Step := ST145_Pnp_e.INIT;
        //Start Manu Ablauf
    ELSIF enIN_State = StateMANU AND xIN_NextStep THEN
        iOUT_Step := ST145_Pnp_e.INIT;
    END_IF;

(***** INIT *****)
ST145_Pnp_e.INIT: (* Grundstellung ? *)
    IF fb_axis145_02Z.xOUT_HOMED THEN
        iOUT_Step := ST145_Pnp_e.Init_VerticalsUp;
    ELSE
        iOUT_Step := ST145_Pnp_e.Init_HomeVerticals;
    END_IF;

ST145_Pnp_e.Init_HomeVerticals:
    IF fb_axis145_02Z.xOUT_HOMED THEN
        iOUT_Step := ST145_Pnp_e.Init_VerticalsUp;
    END_IF

ST145_Pnp_e.Init_VerticalsUp:
    IF fb_vakumGriperLeft.xIN_AS OR fb_vakumGriperRight.xIN_AS THEN
        IF fb_PnpVerAxis.MoveTo(ST145_PnpVerPos_e.UpFull).xOUT_InPos THEN
            IF fb_axis145_01Y.xOUT_HOMED THEN
                iOUT_Step := ST145_Pnp_e.Init_HorizontalsToTrack;
            ELSE
                iOUT_Step := ST145_Pnp_e.Init_HomeHorizontals;
            END_IF
        END_IF
    ELSE
        IF fb_PnpVerAxis.MoveTo(ST145_PnpVerPos_e.UpEmpty).xOUT_InPos THEN
            IF fb_axis145_01Y.xOUT_HOMED THEN
                iOUT_Step := ST145_Pnp_e.Init_HorizontalsToTrack;
            ELSE
                iOUT_Step := ST145_Pnp_e.Init_HomeHorizontals;
            END_IF
        END_IF
    END_IF

ST145_Pnp_e.Init_HomeHorizontals:
    IF fb_axis145_01Y.xOUT_HOMED THEN
        iOUT_Step := ST145_Pnp_e.Init_HorizontalsToTrack;
    END_IF

ST145_Pnp_e.Init_HorizontalsToTrack:
    fb_axis145_02Z.rIN_Velocity := ST145_Axis.const145_02Z.VELO_MANU;

    IF fb_PnpHorAxis.MoveTo(ST145_PnpHorPos_e.GS_Before_placement).xOUT_InPos THEN
        iOUT_Step := ST145_Pnp_e.Init_check_if_pces_handled;
    END_IF

ST145_Pnp_e.Init_check_if_pces_handled:
    IF (NOT _20_AUTO.recipe.st145.xUseVerLeft AND fb_vakumGriperLeft.xOUT_inAS) OR
       (NOT _20_AUTO.recipe.st145.xUseVerRight AND fb_vakumGriperRight.xOUT_inAS) THEN
        // ERROR: a piece is present in an unused gripper
        bOUT_Error := 1;
        iOUT_Step  := ST145_Pnp_e.ERROR;

    ELSIF _20_AUTO.recipe.st145.xUseVerLeft AND
          NOT fb_vakumGriperLeft.xOUT_inAS AND
          _20_AUTO.recipe.st145.xUseVerRight AND
          fb_vakumGriperRight.xOUT_inAS THEN
        // ERROR:  Initialisation failed. A piece is missing in the left griper.
        bOUT_Error := 2;
        iOUT_Step  := ST145_Pnp_e.ERROR;

    ELSIF _20_AUTO.recipe.st145.xUseVerLeft AND
          fb_vakumGriperLeft.xOUT_inAS AND
          _20_AUTO.recipe.st145.xUseVerRight AND
          NOT fb_vakumGriperRight.xOUT_inAS THEN
        // ERROR:  Initialisation failed. A piece is missing in the right griper.
        bOUT_Error := 3;
        iOUT_Step  := ST145_Pnp_e.ERROR;

    ELSIF NOT fb_vakumGriperLeft.xOUT_inAS AND NOT fb_vakumGriperRight.xOUT_inAS THEN
        iOUT_Step := ST145_Pnp_e.READY;

    ELSE
        iOUT_Step := ST145_Pnp_e.waitOnMover;
    END_IF

(***** READY / INIT DONE *****)
ST145_Pnp_e.READY:    (* Start AUTO,END,LEER,STEP *)
    IF xIN_Start THEN //IF rtSTART.Q THEN
        iOUT_Step := ST145_Pnp_e.START;
        iPreStep  := ST145_Pnp_e.INIT;
    END_IF

(***** START  ZYKLISCH *****)
ST145_Pnp_e.START: (*  *)
    IF xIN_NextStep AND pxFG_Freigabe^ THEN
        IF enState.StateLEER = enIN_State THEN
            IF __ISVALIDREF(Mover) THEN
                IF Mover.GetLastStationDone() > 0 THEN
                    iOUT_Step := ST145_Pnp_e.Pnp_Hor_ToRotTablePos;
                ELSE
                    iOUT_Step := ST145_Pnp_e.waitOnMover;
                END_IF
            END_IF
        ELSE
            iOUT_Step := ST145_Pnp_e.Pnp_Hor_ToRotTablePos;
        END_IF
    END_IF;

ST145_Pnp_e.Pnp_Hor_ToRotTablePos:
    IF xIN_NextStep AND fb_PnpHorAxis.MoveTo(ST145_PnpHorPos_e.AS_to_feeder).xOUT_InPos THEN
        iOUT_Step := ST145_Pnp_e.Pnp_WaitOnFeeder;
    END_IF

ST145_Pnp_e.Pnp_WaitOnFeeder:
    IF xIN_PceReadyToPick THEN
        iOUT_Step := ST145_Pnp_e.Pnp_Ver_RotTableDown;
    END_IF

ST145_Pnp_e.Pnp_Ver_RotTableDown:
    IF xIN_NextStep AND fb_PnpVerAxis.MoveTo(ST145_PnpVerPos_e.DownEmpty).xOUT_InPos THEN
        iOUT_Step := ST145_Pnp_e.Vacum_on;
    END_IF;

ST145_Pnp_e.Vacum_on:
    IF xIN_NextStep AND
       (NOT _20_AUTO.recipe.st145.xUseVerLeft OR fb_vakumGriperLeft.xOUT_inAS) AND
       (NOT _20_AUTO.recipe.st145.xUseVerRight OR fb_vakumGriperRight.xOUT_inAS) THEN
        iOUT_Step := ST145_Pnp_e.Pnp_Ver_RotTableUp;
    END_IF;

ST145_Pnp_e.Pnp_Ver_RotTableUp:
    IF xIN_NextStep AND fb_PnpVerAxis.MoveTo(ST145_PnpVerPos_e.UpFull).xOUT_InPos THEN
        iOUT_Step := ST145_Pnp_e.Pnp_Hor_ToTrackPos;
    END_IF;

ST145_Pnp_e.Pnp_Hor_ToTrackPos:
    IF xIN_NextStep AND fb_PnpHorAxis.MoveTo(ST145_PnpHorPos_e.GS_Before_placement).xOUT_InPos THEN
        iOUT_Step := ST145_Pnp_e.waitOnMover;
    END_IF

ST145_Pnp_e.waitOnMover: (*  *)
    IF xIN_NextStep AND __ISVALIDREF(Mover) OR HMI.bArForceCyclusState[StationList_e.ST145] THEN
        IF Mover.GetLastStationDone() >= INT#145 THEN
            iOUT_Step := ST145_Pnp_e.SYNC_MOVER_LEAVE;
        ELSIF Mover.GetLastStationDone() < INT#130 THEN
            iOUT_Step := ST145_Pnp_e.SYNC_MOVER_LEAVE;
        ELSE
            iOUT_Step := ST145_Pnp_e.Pnp_Ver_ShuttleDown;
        END_IF
    END_IF;

ST145_Pnp_e.Pnp_Ver_ShuttleDown:
    IF xIN_NextStep AND fb_PnpVerAxis.MoveTo(ST145_PnpVerPos_e.DownFullQuick).xOUT_InPos THEN
        iOUT_Step := ST145_Pnp_e.Vacum_off;

        IF __ISVALIDREF(Mover) THEN
            IF NOT Mover.SetLastStation(145) THEN
                ASSERT(0);
            END_IF
        END_IF
    END_IF;

// not used here, maybe later
ST145_Pnp_e.Pnp_Ver_ShuttleTorqueControl:
    ASSERT(0);
    iOUT_Step := ST145_Pnp_e.Vacum_off;

ST145_Pnp_e.Vacum_off:
    IF xIN_NextStep AND
       (NOT _20_AUTO.recipe.st145.xUseVerLeft OR fb_vakumGriperLeft.xOUT_inGS) AND
       (NOT _20_AUTO.recipe.st145.xUseVerRight OR fb_vakumGriperRight.xOUT_inGS) THEN
        iOUT_Step := ST145_Pnp_e.Pnp_move_a_bit_to_feeder;
    END_IF

ST145_Pnp_e.Pnp_move_a_bit_to_feeder:
    IF xIN_NextStep AND fb_PnpHorAxis.MoveTo(ST145_PnpHorPos_e.GS_After_placement).xOUT_InPos THEN
        iOUT_Step := ST145_Pnp_e.PnP_Ver_ShuttleUp;
    END_IF

ST145_Pnp_e.PnP_Ver_ShuttleUp:
    IF xIN_NextStep AND fb_PnpVerAxis.MoveTo(ST145_PnpVerPos_e.UpEmpty).xOUT_InPos THEN
        iOUT_Step := ST145_Pnp_e.SYNC_MOVER_LEAVE;

        IF __ISVALIDREF(Mover) THEN
            IF NOT Mover.SetLastStation(145) THEN
                ASSERT(0);
            END_IF
        END_IF
    END_IF;

ST145_Pnp_e.SYNC_MOVER_LEAVE:
    // The mover needs to be taken by MoverMan
    IF NOT __ISVALIDREF(Mover) THEN
        IF (NOT _20_AUTO.recipe.st145.xUseVerLeft OR fb_vakumGriperLeft.xOUT_inAS) AND
           (NOT _20_AUTO.recipe.st145.xUseVerRight OR fb_vakumGriperRight.xOUT_inAS) THEN
            iOUT_Step := ST145_Pnp_e.waitOnMover;
        ELSE
            iOUT_Step := ST145_Pnp_e.DONE;
        END_IF
    END_IF

(***** DONE *****)
ST145_Pnp_e.DONE: (* Letzter Schritt  *)
    IF NOT xIN_AlarmAktiv THEN
        //AUTO
        IF (enIN_State = StateAUTO) AND xIN_RestartCYCL THEN
            iOUT_Step := ST145_Pnp_e.START;
            //STEP / END / LEERFAHREN restart
        ELSIF (enIN_State < StateAUTO) AND (enIN_State >= enState.StateSTEP) AND xIN_RestartCYCL THEN
            iOUT_Step := ST145_Pnp_e.START;
            //STEP / END / LEERFAHREN fertig
        ELSIF (enIN_State = StateREADY) THEN
            iOUT_Step := ST145_Pnp_e.READY;
        END_IF;
    END_IF;

(************ ERROR *************)
ST145_Pnp_e.ERROR: (* ERROR *) ;

END_CASE;

END_FUNCTION_BLOCK

// ---- POUs/20_AUTO/ST145/FB_ABL_145_Feeder.TcPOU
FUNCTION_BLOCK FB_ABL_145_Feeder
(****************************************************************************************)
(*	TITEL				RFID-Ring laden, Feeder and rotary table                        *)
(*	Status				ungetestet                         								*)
(*	Beschrieb:			Ablaufbeschreibung												*)
(*																						*)
(*	Steps:	self-explained using enum													*)
(***********************************Revisionen*******************************************)
(*	see github blames																	*)
(****************************************************************************************)

VAR_INPUT
    xIN_Reset       : BOOL;          // Schrittkette zurücksetzen 
    xIN_Init        : BOOL;          // Initialisieren
    xIN_Quit        : BOOL;          // Fehler quittieren 
    xIN_Start       : BOOL;          // Startbefehl
    xIN_Sperre      : BOOL;          // FB Sperren 
    xIN_NextStep    : BOOL;          // Nächsten Schritt ausführen 
    xIN_AlarmAktiv  : BOOL;          // Anlage hat Alarm
    xIN_DryCycle    : BOOL;          // Fahren ohne Teile
    xIN_RestartCYCL : BOOL;          // Zyklus erneut starten im STEP, END, LEERFAHREN
    enIN_State      : enState;       // Status Anlage
    tIN_Timeout     : TIME := T#10s; // Timout

    pxFG_Freigabe : POINTER TO BOOL; //Freigabe von Station

    // Application specific
    xIN_PickPiece : BOOL; (* signal from the pick and place element
                             the number of picked signal depend on the recipe *)
    xIN_RotTableBlockedByPnp : BOOL; // Is the pick and place blocking the rotary table?
END_VAR
VAR_OUTPUT
    (* standart Ausgänge *)
    xOUT_ErrFlag  : BOOL;           // Error Flag 
    xOUT_Busy     : BOOL;           // Baustein befindet sich im Ablauf 
    xOUT_Done     : BOOL;           // Baustein hat den Ablauf beendet 		
    xOUT_Ready    : BOOL;           // Ready to begin, should be the same state as done	
    xOUT_Timeout  : BOOL;           // Timeout FB 
    xOUT_InitDone : BOOL;           // initialisierung fertig
    xOUT_Wait     : BOOL;           // Wartet auf Bedingung
    iOUT_Step     : ST145_Feeder_e; // Aktueller Schritt 
    sOUT_Step     : STRING;         // Aktueller Schritt but in string format
    bOUT_Error    : BYTE;           // Fehlernummer

    // Application specific
    xOUT_PceReadyToPick : BOOL; // the piece(s) is/are ready to picked
END_VAR
VAR
    (* Standard *)
    (* Schritt *)
    iLastStep : ST145_Feeder_e; // Merker letzter Schritt 
    iPreStep  : ST145_Feeder_e; // Schritt zurück nach Alarm 
    iAktStep  : ST145_Feeder_e; // aktueller Schritt

    // Trigger Starten 
    rtSTART : R_TRIG;
    // Timer TimeOut 
    TON_Timeout : TON;

    (* Bausteine *)

    // Application specific
    fb_axis145_10W               : FB_AxisLMturn_V1_1;
    simu_axis145_10W             : FB_Simu_AxisLM_V1_1;
    fb_feeder                    : FB_Feeder2Sensors;
    fifo                         : FB_Fifo(3);
    simu_feeder                  : FB_Simu_Feeder; // simulation of a feeder
    simu_fifo_feeder_to_rotTable : FB_Fifo(20);    // fifo to hold a piece
    rtPutPiece                   : R_TRIG;         // trigger to add a piece

    rtPick : R_TRIG; // r_trig signal from the pick and place machine

    iCurrentTableIndex : INT; // current table index
    iSearchIndex       : INT; (* Initialization index TO see how many element we have AT startup
                                 or after an alarm *)

END_VAR
VAR CONSTANT
    MAX_SEARCH_TURN : INT := 3; // maximum search number

    FEEDER_SIMULATION : BOOL := FALSE; // Simulate this code
END_VAR

(*******************************************************************)
(* Trigger  *)
(*******************************************************************)
(* Zurücksetzen *)
IF xIN_RESET THEN
    iPreStep  := ST145_Feeder_e.RESET;
    iOUT_Step := ST145_Feeder_e.RESET;
END_IF;

(* Error Quittieren *)
IF (bOUT_Error <> 0) AND xIN_Quit THEN
    xOUT_ErrFlag := FALSE;
    bOUT_Error   := 0;
    iOUT_Step    := iPreStep;
END_IF;

iCurrentTableIndex := iCurrentTableIndex MOD 3;

(*******************************************************************)
(* Timer *)
(*******************************************************************)
TON_Timeout(IN := xIN_NextStep AND (iLastStep = iOUT_Step) (*todo FG *) ,
            PT := tIN_Timeout);

(*******************************************************************)
(* Bausteine *)
(*******************************************************************)
fb_feeder(xIN_Enable                := enIN_State = enState.StateAUTO OR enIN_State = enState.StateSTEP,
          xIN_PieceInEnd            := IO_BOX.I2401_ST145_maximum_wf,
          xIN_PieceMax              := IO_BOX.I2401_ST145_maximum_wf,
          xIN_InSimulation          := FEEDER_SIMULATION AND CONST.USE_SIMULATION,
          refIN_SimulatedFifo       := simu_fifo_feeder_to_rotTable,
          iIN_FifoSetMaxSensorValue := 10,
          diIN_SignlFilter_ms       := _20_AUTO.recipe.st145.FeederConfig.InFilterDelay,
          diIN_StartDelay_ms        := _20_AUTO.recipe.st145.FeederConfig.StartDelay,
          diIN_StopDelay_ms         := _20_AUTO.recipe.st145.FeederConfig.StopDelay,
          diIN_EmptyDelay_ms        := _20_AUTO.recipe.st145.FeederConfig.EmptyDelay);

simu_feeder(xIN_Enable         := fb_feeder.xOUT_EnableFeeder AND FEEDER_SIMULATION AND CONST.USE_SIMULATION,
            xIN_PceSensor      := IO_BOX.I2300_ST145_teil_in_vereinzelung,
            tIN_NewPieceTime   := 500,
            iIN_WaitTimeMin_ms := 500,
            iIN_WaitTimeMax_ms := 1000);

rtPick(CLK := xIN_PickPiece);
rtPutPiece(CLK := simu_feeder.xOUT_NewPiece);

IF rtPutPiece.Q AND NOT simu_fifo_feeder_to_rotTable.IsFull() THEN
    simu_fifo_feeder_to_rotTable.Put(1);
END_IF

IF ST145_Feeder_e.Init_simu_home_table = iOUT_Step THEN
    fb_axis145_10W.rIN_Position := TO_REAL(120.0 - LMOD(ST145_Axis.axis145_10W.rActPos, 120.0));

ELSIF ST145_Feeder_e.Init_home_table = iOUT_Step THEN
    fb_axis145_10W.rIN_Position := TO_REAL(120.0 - LMOD(ST145_Axis.axis145_10W.rActPos, 120.0));

ELSIF ST145_Feeder_e.Init_table_go_to_zero = iOUT_Step THEN
    fb_axis145_10W.rIN_Position := 360 - ST145_Axis.axis145_10W.rActPos;

ELSE
    fb_axis145_10W.rIN_Position := 120.0;

END_IF

simu_axis145_10W(xIN_Enable          := FEEDER_SIMULATION AND CONST.USE_SIMULATION,
                 wIN_AxisState       := ST145_Axis.axis145_10W.wState,
                 bIN_AxisCntr        := fb_axis145_10W.bOUT_AxisCntr,
                 udiIN_HomingTime_ms := 1000,
                 pIN_axisSimu        := ADR(SIMU.axis_ref[Axis_e.ST145_10W]),
                 pIN_axisHW          := ADR(ST145_Axis.axis145_10W.axis),
                 rIN_PosActual       := fb_axis145_10W.rOUT_ActPos,
                 rIN_PosMax          := ST145_Axis.const145_10W.POS_MAX,
                 rIN_PosMin          := ST145_Axis.const145_10W.POS_MIN,
                 rIN_PixMax          := 0,
                 rIN_PixMin          := 0);

fb_axis145_10W(enIN_State     := enIN_State,
               parIN_Buttons  := ADR(AXIS.btTeachArAxis[Axis_e.ST145_10W]),
               xIN_DisButtons :=,
               xIN_Quit       := xIN_Quit,
               xIN_PARAMok    := TRUE,
               xIN_FREE       := TRUE,
               xIN_FREE_HOME  := TRUE,
               rIN_POSMIN     := ST145_Axis.const145_10W.POS_MIN,
               rIN_POSMAX     := ST145_Axis.const145_10W.POS_MAX,
               rIN_VELOMAX    := ST145_Axis.const145_10W.VELO_MAX,
               rIN_VELOMANU   := ST145_Axis.const145_10W.VELO_MANU,
               rIN_VELOOPEN   := ST145_Axis.const145_10W.VELO_MANU / 4,
               rIN_JogInc     := AXIS.rTeachIncAxis,
               xIN_Execute    := ST145_Feeder_e.Init_set_table_pos = iOUT_Step OR
                                 ST145_Feeder_e.Init_table_go_to_zero = iOUT_Step OR
                                 ST145_Feeder_e.Init_simu_home_table = iOUT_Step OR
                                 ST145_Feeder_e.load_piece = iOUT_Step OR
                                 ST145_Feeder_e.wait_rotary_table_done = iOUT_Step,
               xIN_Relative     := TRUE,
               xIN_STOP         := FALSE,
               xIN_OFF          := FALSE,
               rIN_Position     :=, // Is set above
               rIN_Velocity     := TO_REAL(100.0),
               rIN_Acceleration := TO_REAL(720.0),
               rIN_Deceleration := TO_REAL(720.0),
               rIN_Jerk         := TO_REAL(72000.0),
               xIN_Home         := ST145_feeder_e.Init_home_table = iOUT_Step,
               xIN_Reset        := xIN_Reset OR ST145_feeder_e.RESET = iOUT_Step,
               // The simu fb gives us the hardware signal when we are not in simulation
               wAxisState    := simu_axis145_10W.wOUT_AxisState,
               bOUT_AxisCntr => ST145_Axis.axis145_10W.bCtrlHi,
               rOUT_ActPos   =>, // leave empty, rActPos must be set using the modulo
               axisIN_REF    := simu_axis145_10W.pOUT_axisRef^);

ST145_Axis.axis145_10W.rActPos := LREAL_TO_REAL(simu_axis145_10W.pOUT_axisRef^.NcToPlc.ModuloActPos);

(*******************************************************************)
(* OUTPUTS *)
(*******************************************************************)
// Error Flag 
xOUT_ErrFlag := (bOUT_Error <> 0) OR (ST145_Feeder_e.ERROR = iOUT_Step);
// Baustein befindet sich im Ablauf 
xOUT_Busy := (iOUT_Step > ST145_Feeder_e.READY) AND (iOUT_Step < ST145_Feeder_e.DONE);
// Baustein hat den Ablauf beendet
xOUT_Done := (iOUT_Step = ST145_Feeder_e.DONE);
// Process ready
xOUT_Ready := (iOUT_Step = ST145_Feeder_e.READY);
// Timeout FB 				 		
xOUT_Timeout := TON_Timeout.Q;
// Itialisierung fertig			
xOUT_InitDone := (iOUT_Step = ST145_Feeder_e.READY);
// Aktueller Schritt			
iOUT_Step := iOUT_Step; //Im Ablauf gesetzt		
sOUT_Step := TO_STRING(iOUT_Step);
//Fehlernummer	 
bOUT_Error := bOUT_Error; //Im Ablauf/FB gesetzt	
(* Warte (alle Schritte wo auf FG oder Teile gewartet wird) *)
xOUT_Wait := (iOUT_Step = ST145_Feeder_e.DONE) OR
             (iOUT_Step = ST145_Feeder_e.READY);

// TODO add simulation constant to prevent the output to be set
IO_BOX.Q2402_ST145_reigabe_wf := fb_feeder.xOUT_EnableFeeder AND
                                 NOT (FEEDER_SIMULATION AND CONST.USE_SIMULATION);

IO_BOX.Q2400_ST145_freigabe_REO := ((iOUT_Step = ST145_Feeder_e.wait_on_a_piece) OR
                                   IO_BOX.Q2402_ST145_reigabe_wf OR
                                   ((iOUT_Step = ST145_Feeder_e.DONE) AND NOT IO_BOX.I2300_ST145_teil_in_vereinzelung)
                                       ) AND
                                   NOT (FEEDER_SIMULATION AND CONST.USE_SIMULATION);

(*******************************************************************)
(* Ablauf *)
(*******************************************************************)

(* Sperren *)
IF xIN_Sperre THEN
    iPreStep  := ST145_Feeder_e.RESET;
    iOUT_Step := ST145_Feeder_e.RESET;
    RETURN;
END_IF;

(* Schritt Merker *)
IF iAktStep <> iOUT_Step THEN
    iLastStep := iAktStep;
    iAktStep  := iOUT_Step;
END_IF

(* START *)
rtSTART(CLK := xIN_Start);

IF 0 = bOUT_Error THEN
    IF fb_axis145_10W.xOUT_ErrFlag THEN
        bOUT_Error := 11;
        iPreStep   := ST145_Feeder_e.RESET;
    END_IF
ELSIF iOUT_Step < ST145_Feeder_e.ERROR THEN
    iOUT_Step := ST145_Feeder_e.ERROR;
END_IF

(*******************************************************************)
(* Schrittkette  *)
(*******************************************************************)
CASE iOUT_Step OF

(***** RESET *****)
ST145_Feeder_e.RESET: (* Schritt 0-99 *)
    //Initialisierungen
    //Start Init Ablauf
    IF xIN_Init THEN
        iOUT_Step := ST145_Feeder_e.INIT;
        //Start Manu Ablauf
    ELSIF enIN_State = StateMANU AND xIN_NextStep THEN
        iOUT_Step := ST145_Feeder_e.INIT;
    END_IF;

(***** INIT *****)
ST145_Feeder_e.INIT: (* Grundstellung ? *)
    IF NOT xIN_RotTableBlockedByPnp THEN
        iOUT_Step := ST145_Feeder_e.Init_home_table;
    END_IF

ST145_Feeder_e.Init_home_table:
    IF fb_axis145_10W.xOUT_HOMED THEN
        iCurrentTableIndex := 0;

        IF FEEDER_SIMULATION AND CONST.USE_SIMULATION THEN
            iOUT_Step := ST145_Feeder_e.Init_simu_home_table;
        ELSE
            iOUT_Step := ST145_Feeder_e.Init_table_go_to_zero;
        END_IF
    END_IF

ST145_Feeder_e.Init_simu_home_table:
    IF fb_axis145_10W.xOUT_DONE THEN
        iOUT_Step := ST145_Feeder_e.Init_reset_search_index;
    END_IF

// unused, zero position is done by the configuration of the drive
ST145_Feeder_e.Init_table_go_to_zero:
    IF fb_axis145_10W.xOUT_DONE THEN
        iOUT_Step := ST145_Feeder_e.Init_reset_search_index;
    END_IF

ST145_Feeder_e.Init_reset_search_index:
    iSearchIndex := 0;
    fifo.Empty();
    iOUT_Step := ST145_Feeder_e.READY; // Bypass search algorithm, unusful

ST145_Feeder_e.Init_set_table_pos:
    IF fb_axis145_10W.xOUT_DONE THEN
        iCurrentTableIndex := iCurrentTableIndex + 1;
        iOUT_Step          := ST145_Feeder_e.Init_see_if_piece_there;
    END_IF

ST145_Feeder_e.Init_see_if_piece_there:
    IF simu_feeder.xOUT_NewPiece THEN
        fifo.Put(1);
    END_IF

    IF iSearchIndex < MAX_SEARCH_TURN THEN
        iOUT_Step    := ST145_Feeder_e.Init_set_table_pos;
        iSearchIndex := iSearchIndex + 1;
    ELSE
        iOUT_Step := ST145_Feeder_e.READY;
    END_IF

(***** READY / INIT DONE *****)
ST145_Feeder_e.READY: (* Start AUTO,END,LEER,STEP *)
    IF xIN_Start THEN //IF rtSTART.Q THEN
        iOUT_Step := ST145_Feeder_e.START;
    END_IF

(***** START  ZYKLISCH *****)
ST145_Feeder_e.START: (*  *)
    IF xIN_NextStep AND pxFG_Freigabe^ THEN
        iOUT_Step := ST145_Feeder_e.check_if_feeding_necessary;
    END_IF;

ST145_Feeder_e.check_if_feeding_necessary:
    IF fifo.IsFull() THEN
        iOUT_Step := ST145_Feeder_e.DONE;
    ELSE
        iOUT_Step := ST145_Feeder_e.wait_on_a_piece;
    END_IF

ST145_Feeder_e.wait_on_a_piece:
    IF (FEEDER_SIMULATION AND CONST.USE_SIMULATION AND NOT simu_fifo_feeder_to_rotTable.IsEmpty()) OR
       (NOT (FEEDER_SIMULATION AND CONST.USE_SIMULATION) AND IO_BOX.I2300_ST145_teil_in_vereinzelung) THEN
        IF NOT xIN_RotTableBlockedByPnp THEN
            iOUT_Step := ST145_Feeder_e.load_piece;
            simu_fifo_feeder_to_rotTable.Pop(1);
        END_IF
    END_IF

ST145_Feeder_e.load_piece:
    IF NOT fb_axis145_10W.xOUT_DONE THEN
        iOUT_Step := ST145_Feeder_e.wait_rotary_table_done;
    END_IF

ST145_Feeder_e.wait_rotary_table_done:
    IF fb_axis145_10W.xOUT_DONE THEN
        fifo.Put(1);
        iOUT_Step := ST145_Feeder_e.check_if_feeding_necessary;
    END_IF

(***** DONE *****)
ST145_Feeder_e.DONE: (* Letzter Schritt  *)
    IF rtPick.Q THEN
        fifo.Pop(TO_INT(_20_AUTO.recipe.st145.xUseVerLeft));
        fifo.Pop(TO_INT(_20_AUTO.recipe.st145.xUseVerRight));
    END_IF

    IF NOT xIN_AlarmAktiv THEN
        //AUTO
        IF (enIN_State = StateAUTO) AND xIN_RestartCYCL AND NOT fifo.IsFull() THEN
            iOUT_Step := ST145_Feeder_e.START;
            //STEP / END / LEERFAHREN restart
        ELSIF (enIN_State < StateAUTO) AND (enIN_State >= enState.StateSTEP) AND xIN_RestartCYCL AND NOT fifo.IsFull()
            THEN
            iOUT_Step := ST145_Feeder_e.START;
            //STEP / END / LEERFAHREN fertig
        ELSIF (enIN_State = StateREADY) THEN
            iOUT_Step := ST145_Feeder_e.READY;
        END_IF;
    END_IF;

(************ ERROR *************)
ST145_Feeder_e.ERROR: (* ERROR *) ;

END_CASE;

END_FUNCTION_BLOCK

// ---- POUs/20_AUTO/ST15x/FB_AUT_150.TcPOU
FUNCTION_BLOCK FB_AUT_150 EXTENDS FB_AUT_ABSTRACT
(****************************************************************************)
(*	POU_AUT_zxx			Bausteinaufrufe Station	zxx							*)
(*	Status				ungetestet											*)
(*  Version:			1.0													*)
(*	Beschrieb:																*)
(*																			*)
(*	Abläufe:			FB_ABLzxxA		Hauptablauf							*)
(*																			*)
(*																			*)
(* 	25.09.2019/Dj															*)
(****************************************************************************)
(*	dd.mm.yyyy   KZ    x.y			Beschrieb								*)
(****************************************************************************)
VAR_INPUT
    (* spezifische Eingänge *)

END_VAR
VAR_OUTPUT
    (* spezifische Ausgänge *)

END_VAR
VAR
    (* Bausteine *)
    fb_Uss : FB_ABL_150;

    fb_stat : FB_AUT_Statistics;

END_VAR

(*******************************************************************)
(* Timer *)
(*******************************************************************)

(*******************************************************************)
(* Flanken / Merker *)
(*******************************************************************)
//MANU CYCLE
IF (enIN_State = StateMANU) AND xIN_ManuCycle THEN
    xManuCycle := TRUE;
END_IF;

IF (enIN_State <> StateMANU) OR xOUT_Done THEN
    xManuCycle := FALSE;
END_IF

//NEXT STEP
xNextStep := (enIN_State > StateSTEP) OR
             ((enIN_State = StateSTEP) AND xIN_Step) OR
             ((enIN_State = StateMANU) AND xManuCycle);

//RESET
xReset := (enIN_State < StateREADY) AND (enIN_State <> StateINIT) AND NOT xManuCycle;

(*******************************************************************)
(* Bausteinaufrufe Abläufe *)
(*******************************************************************)

xRelease := MAIN.MoverMan.IsProcessUsed(THIS^);

fb_Uss.xIN_welding_bits.Bereit       := IN.I020_ultraschall_bereit_150_20;
fb_Uss.xIN_welding_bits.Fehler       := IN.I021_ultraschall_fehler_150_20;
fb_Uss.xIN_welding_bits.US_on        := IN.I022_ultraschall_us_on_150_20;
fb_Uss.xIN_welding_bits.NullPosition := IN.I023_ultraschall_nullpos_150_20;

fb_Uss(xIN_Reset       := xReset,
       xIN_Init        := xIN_Init,
       xIN_Quit        := xIN_Quit,
       xIN_Start       := enIN_State >= enState.StateLEER AND xRelease,
       xIN_Sperre      := NOT xIN_On,
       xIN_NextStep    := xNextStep,
       xIN_AlarmAktiv  := xIN_AlarmAktiv,
       xIN_DryCycle    := xIN_DryCycle,
       xIN_RestartCYCL := enIN_State >= enState.StateLEER,
       enIN_State      := enIN_State,
       tIN_Timeout     := tIN_Timeout,
       pxFG_Freigabe   := ADR(xRelease),
       // CleverTrackLib
       Mover := THIS^.Mover,
       // hardware input
       xIN_capDetector             := IO_BOX.I2303_ST150_deckel_vohanden,
       xIN_kraftubersetzunh_zuruck := IO_BOX.I2301_ST150_kraftubersetzung_zuruck,
       xIN_kraftubersetzunh_vor    := IO_BOX.I2302_ST150_kraftubersetzung_vor,
       pIN_ButtonMaintaining       := ADR(HMI.btManuCylinders[StationList_e.ST150][1]),
       xIN_welding_bits            :=, // set above
       iIN_StationNumber           := 150,
       sIN_errorCodeSide           := 'Left',
       // hardware output
       xOUT_moverMaintening_valve => IO_BOX.Q0202_14_ST150_kraftubersetzung,
       xOUT_welding_bits          =>); // set below

OUT.Q020_ST150_ultraschall_start      := fb_Uss.xOUT_welding_bits.Start;
OUT.Q021_ST150_ultraschall_reset      := fb_Uss.xOUT_welding_bits.Reset;
OUT.Q022_ST150_ultraschall_data_bit_0 := fb_Uss.xOUT_welding_bits.Data_Hex1;
OUT.Q023_ST150_ultraschall_data_bit_1 := fb_Uss.xOUT_welding_bits.Data_Hex2;
OUT.Q024_ST150_ultraschall_data_bit_2 := fb_Uss.xOUT_welding_bits.Data_Hex4;
OUT.Q025_ST150_ultraschall_data_bit_3 := fb_Uss.xOUT_welding_bits.Data_Hex8;

fb_stat(xIN_Enable  := enState.StateAUTO = enIN_State,
        xIN_Waiting := fb_Uss.xOUT_Wait,
        xIN_Running := (fb_Uss.iOUT_Step >= ST150_Uss_e.START) AND
                       (fb_Uss.iOUT_Step <= ST150_Uss_e.DONE),
        // Since we use a mover system, a cycle is done when we are waiting on a mover
        xIN_Done := fb_Uss.iOUT_Step = ST150_Uss_e.waitOnMover);

(*******************************************************************)
(* Mover reset flags *)
(*******************************************************************)

(*******************************************************************)
(* OUTPUT *)
(*******************************************************************)
xOUT_InitDone := fb_Uss.xOUT_InitDone;
xOUT_Ready    := fb_Uss.xOUT_Ready;
xOUT_Done     := fb_Uss.xOUT_Done;
xOUT_ErrFlag  := fb_Uss.xOUT_ErrFlag;
xOUT_Wait     := fb_Uss.xOUT_Wait;
xOUT_AlarmST  := xOUT_ErrFlag;

(*******************************************************************)
(* Bausteinaufruf Error Station *)
(*******************************************************************)
// POU_ERR_VORLAGE(xIN_QUIT:=xIN_Quit , pstrArIN_ALARM:=ADR(HMI.strArALARM[1]));

(* % of completion of the process *)
PROPERTY iCompletionPC : INT
GET
iCompletionPC := THIS^.fb_Uss.iOUT_ProcessCompletion;
END_GET
END_PROPERTY

PROPERTY ProcessExecution : ProcessExecution_e
GET
ProcessExecution := THIS^._ProcessExecution;
END_GET
SET
THIS^._ProcessExecution := ProcessExecution;
END_SET
END_PROPERTY

PROPERTY xBusy : BOOL
GET
xBusy := THIS^.fb_Uss.xOUT_Busy;
END_GET
SET
END_SET
END_PROPERTY

PROPERTY xDone : BOOL
GET
xDone := THIS^.fb_Uss.xOUT_Ready OR THIS^.fb_Uss.xOUT_Done;
END_GET
END_PROPERTY

PROPERTY xMoverPathFree : BOOL
GET
xMoverPathFree := THIS^.fb_Uss.xOUT_MoverFree OR THIS^.fb_Uss.xOUT_Ready OR THIS^.fb_Uss.xOUT_Done;
END_GET
END_PROPERTY

PROPERTY xMoverShouldLeave : BOOL
GET
xMoverShouldLeave := THIS^.fb_Uss.iOUT_Step = ST150_Uss_e.SYNC_MOVER_LEAVE;
END_GET
END_PROPERTY

END_FUNCTION_BLOCK

// ---- POUs/20_AUTO/ST15x/FB_ABL_150.TcPOU
FUNCTION_BLOCK FB_ABL_150
(****************************************************************************************)
(*	TITEL				laden kristall- Modul	    										*)
(*	Status				ungetestet                         								*)
(*	Beschrieb:			Ablaufbeschreibung												*)
(*																						*)
(*	Steps:	self-explained using enum													*)
(***********************************Revisionen*******************************************)
(*	see github blames																	*)
(****************************************************************************************)

VAR_INPUT
    xIN_Reset       : BOOL;          // Schrittkette zurücksetzen 
    xIN_Init        : BOOL;          // Initialisieren
    xIN_Quit        : BOOL;          // Fehler quittieren 
    xIN_Start       : BOOL;          // Startbefehl
    xIN_Sperre      : BOOL;          // FB Sperren 
    xIN_NextStep    : BOOL;          // Nächsten Schritt ausführen 
    xIN_AlarmAktiv  : BOOL;          // Anlage hat Alarm
    xIN_DryCycle    : BOOL;          // Fahren ohne Teile
    xIN_RestartCYCL : BOOL;          // Zyklus erneut starten im STEP, END, LEERFAHREN
    enIN_State      : enState;       // Status Anlage
    tIN_Timeout     : TIME := T#10s; // Timout

    pxFG_Freigabe : POINTER TO BOOL; //Freigabe von Station

    // Application specific
    Mover : REFERENCE TO FB_Mover;

    xIN_capDetector             : BOOL;
    xIN_kraftubersetzunh_zuruck : BOOL;
    xIN_kraftubersetzunh_vor    : BOOL;

    xIN_welding_bits : Ultrasonic_IN_bits_t;

    iIN_StationNumber : INT;    // station number 
    sIN_errorCodeSide : STRING; // added string to the error code, (e.g. left or right)

END_VAR
VAR_OUTPUT
    (* standart Ausgänge *)
    xOUT_ErrFlag  : BOOL;        // Error Flag 
    xOUT_Busy     : BOOL;        // Baustein befindet sich im Ablauf 
    xOUT_Done     : BOOL;        // Baustein hat den Ablauf beendet 		
    xOUT_Ready    : BOOL;        // Ready to begin, should be the same state as done	
    xOUT_Timeout  : BOOL;        // Timeout FB 
    xOUT_InitDone : BOOL;        // initialisierung fertig
    xOUT_Wait     : BOOL;        // Wartet auf Bedingung
    iOUT_Step     : ST150_Uss_e; // Aktueller Schritt 
    sOUT_Step     : STRING;      // Aktueller Schritt but in string format
    bOUT_Error    : BYTE;        // Fehlernummer

    iOUT_ProcessCompletion : INT;  //process completion, express in % (0-100)
    xOUT_MoverFree         : BOOL; // The mover is free to move

    xOUT_moverMaintening_valve : BOOL;
    xOUT_welding_bits          : Ultrasonic_OUT_bits_t;

END_VAR
VAR
    (* Standard *)
    (* Schritt *)
    iLastStep : ST150_Uss_e; // Merker letzter Schritt 
    iPreStep  : ST150_Uss_e; // Schritt zurück nach Alarm 
    iAktStep  : ST150_Uss_e; // aktueller Schritt

    // Trigger Starten 
    rtSTART : R_TRIG;
    // Timer TimeOut 
    TON_Timeout : TON;

    (* Bausteine *)

    (* Spezial *)
    fb_moverMaintening   : FB_ZylMo2El_V2_1;
    simu_moverMaintening : FB_Simu_Zyl2Pos;

    TON_UssError     : TON;
    TON_CapDetection : TON;

END_VAR
VAR CONSTANT
    USS_SIMULATION : BOOL := FALSE; // Set to TRUE to simulate this part of the program
END_VAR

(*******************************************************************)
(* Trigger  *)
(*******************************************************************)
(* Zurücksetzen *)
IF xIN_RESET THEN
    iPreStep  := ST150_Uss_e.RESET;
    iOUT_Step := ST150_Uss_e.RESET;
END_IF;

(* Error Quittieren *)
IF (bOUT_Error <> 0) AND xIN_Quit THEN
    xOUT_ErrFlag := FALSE;
    bOUT_Error   := 0;
    iOUT_Step    := iPreStep;
END_IF;

(*******************************************************************)
(* Timer *)
(*******************************************************************)
TON_Timeout(IN := xIN_NextStep AND (iLastStep = iOUT_Step) (*todo FG *) ,
            PT := tIN_Timeout);

TON_UssError(IN := ST150_Uss_e.uss_start = iOUT_Step,
             PT := DINT_TO_TIME(_20_AUTO.recipe.st150.USS_ErrorTime_ms));

TON_CapDetection(IN := ST150_Uss_e.check_cap_present = iOUT_Step,
                 PT := T#500MS);

(*******************************************************************)
(* Bausteine *)
(*******************************************************************)
fb_moverMaintening(xIN_Reset    := xIN_Reset OR (ST150_Uss_e.RESET = iOUT_Step),
                   xIN_Quit     := xIN_Quit,
                   xIN_Manu     := enState.StateMANU = enIN_State,
                   pbtIN_Button := ADR(HMI.btManuCylinders[StationList_e.ST150][1]),
                   xIN_GS       := simu_moverMaintening.xOUT_inGS,
                   xIN_AS       := simu_moverMaintening.xOUT_inAS,
                   xIN_FREE     := TRUE,
                   xINtoGS      := (ST150_Uss_e.Init_ResetUss_maintaining_down = iOUT_Step) OR
                                   (ST150_Uss_e.mover_maintening_down = iOUT_Step),
                   xINtoAS   := ST150_Uss_e.mover_maintening_up = iOUT_Step,
                   tIN_ErrAS := DINT_TO_TIME(_20_AUTO.recipe.cylinder2Pos[StationList_e.ST150]
                                                 [ST150_Cylinders_e.Kraftbstutzung].toAS_alarm_time),
                   tIN_ErrGS := DINT_TO_TIME(_20_AUTO.recipe.cylinder2Pos[StationList_e.ST150]
                                                 [ST150_Cylinders_e.Kraftbstutzung].toGS_alarm_time),
                   tIN_WaitAS := DINT_TO_TIME(_20_AUTO.recipe.cylinder2Pos[StationList_e.ST150]
                                                  [ST150_Cylinders_e.Kraftbstutzung].toAS_wait_time),
                   tIN_WaitGS := DINT_TO_TIME(_20_AUTO.recipe.cylinder2Pos[StationList_e.ST150]
                                                  [ST150_Cylinders_e.Kraftbstutzung].toGS_wait_time));

simu_moverMaintening(xIN_Enable := USS_SIMULATION AND CONST.USE_SIMULATION,
                     xIN_inGS   := xIN_kraftubersetzunh_zuruck,
                     xIN_inAS   := xIN_kraftubersetzunh_vor,
                     xIN_valve  := fb_moverMaintening.xOUT_VALVE,
                     tIN_GS_ms  := 200,  // ms
                     tIN_AS_ms  := 200); // ms

(*******************************************************************)
(* OUTPUTS *)
(*******************************************************************)
// Error Flag 
xOUT_ErrFlag := (bOUT_Error <> 0) OR (ST150_Uss_e.ERROR = iOUT_Step);
// Baustein befindet sich im Ablauf 
xOUT_Busy := (iOUT_Step > ST150_Uss_e.READY) AND (iOUT_Step < ST150_Uss_e.DONE);
// Baustein hat den Ablauf beendet
xOUT_Done := (iOUT_Step = ST150_Uss_e.DONE);
// Process ready
xOUT_Ready := (iOUT_Step = ST150_Uss_e.READY) OR (iOUT_Step = ST150_Uss_e.waitOnMover);
// Timeout FB 				 		
xOUT_Timeout := TON_Timeout.Q;
// Itialisierung fertig			
xOUT_InitDone := (iOUT_Step = ST150_Uss_e.READY) OR (iOUT_Step = ST150_Uss_e.waitOnMover);
// Aktueller Schritt			
iOUT_Step := iOUT_Step; //Im Ablauf gesetzt		
sOUT_Step := TO_STRING(iOUT_Step);
//Fehlernummer	 
bOUT_Error := bOUT_Error; //Im Ablauf/FB gesetzt	
(* Warte (alle Schritte wo auf FG oder Teile gewartet wird) *)
xOUT_Wait := (iOUT_Step = ST150_Uss_e.DONE) OR
             (iOUT_Step = ST150_Uss_e.READY) OR
             (iOUT_Step = ST150_Uss_e.START) OR
             (iOUT_Step = ST150_Uss_e.waitOnMover) OR
             (iOUT_Step = ST150_Uss_e.SYNC_MOVER_LEAVE);

xOUT_MoverFree :=
    NOT (iOUT_Step >= ST150_Uss_e.MOVER_NEEDED_OP AND iOUT_Step < ST150_Uss_e.MOVER_FREE_OP) AND
    (iOUT_Step >= ST150_Uss_e.READY) AND
    (iOUT_Step < ST150_Uss_e.ERROR);

iOUT_ProcessCompletion := F_GetPercent_2(iAktStep,
                                         iAktStep,
                                         iAktStep,
                                         ST150_Uss_e.check_cap_present,
                                         ST150_Uss_e.SYNC_MOVER_LEAVE);

xOUT_moverMaintening_valve :=
    fb_moverMaintening.xOUT_VALVE AND NOT (USS_SIMULATION AND CONST.USE_SIMULATION);

xOUT_welding_bits.Start :=
    (ST150_Uss_e.uss_start = iOUT_Step) AND
    NOT (USS_SIMULATION AND CONST.USE_SIMULATION) AND
    xIN_capDetector;

xOUT_welding_bits.Reset :=
    (_14_STATE._FB_btQUIT.pbtIN^.press AND
    NOT (ST150_Uss_e.uss_working = iOUT_Step) AND
    NOT (ST150_Uss_e.uss_start = iOUT_Step)) OR
    (ST150_Uss_e.Init_ResetUss_maintaining_down = iOUT_Step);

xOUT_welding_bits.Data_Hex1 := _20_AUTO.recipe.st150.USS_Type.0; // _20_AUTO.recipe.st150.USS_Type = 1;
xOUT_welding_bits.Data_Hex2 := _20_AUTO.recipe.st150.USS_Type.1; // _20_AUTO.recipe.st150.USS_Type = 2;
xOUT_welding_bits.Data_Hex4 := _20_AUTO.recipe.st150.USS_Type.2; // _20_AUTO.recipe.st150.USS_Type = 3;
xOUT_welding_bits.Data_Hex8 := _20_AUTO.recipe.st150.USS_Type.3; // _20_AUTO.recipe.st150.USS_Type = 4;

(*******************************************************************)
(* Ablauf *)
(*******************************************************************)

(* Sperren *)
IF xIN_Sperre THEN
    iPreStep  := ST150_Uss_e.RESET;
    iOUT_Step := ST150_Uss_e.RESET;
    RETURN;
END_IF;

(* Schritt Merker *)
IF iAktStep <> iOUT_Step THEN
    iLastStep := iAktStep;
    iAktStep  := iOUT_Step;
END_IF

(* START *)
rtSTART(CLK := xIN_Start);

IF 0 = bOUT_Error THEN
    IF fb_moverMaintening.xOUT_ErrFlag THEN
        bOUT_Error := 11;
    ELSIF USS_SIMULATION AND CONST.USE_SIMULATION AND xIN_welding_bits.Fehler THEN
        bOUT_Error := 12;
    ELSIF TON_UssError.Q THEN
        bOUT_Error := 13;
    END_IF
ELSIF iOUT_Step < ST150_Uss_e.ERROR THEN
    iOUT_Step := ST150_Uss_e.ERROR;
END_IF

(*******************************************************************)
(* Schrittkette  *)
(*******************************************************************)
CASE iOUT_Step OF

(***** RESET *****)
ST150_Uss_e.RESET: (* Schritt 0-99 *)
    //Initialisierungen
    //Start Init Ablauf
    IF xIN_Init THEN
        iOUT_Step := ST150_Uss_e.INIT;
        //Start Manu Ablauf
    ELSIF enIN_State = StateMANU AND xIN_NextStep THEN
        iOUT_Step := ST150_Uss_e.INIT;
    END_IF;

(***** INIT *****)
ST150_Uss_e.INIT: (* Grundstellung ? *)
    iOUT_Step := ST150_Uss_e.Init_ResetUss_maintaining_down;

ST150_Uss_e.Init_ResetUss_maintaining_down:
    IF fb_moverMaintening.xOUT_inGS THEN
        iOUT_Step := ST150_Uss_e.READY;
    END_IF

(***** READY / INIT DONE *****)
ST150_Uss_e.READY:    (* Start AUTO,END,LEER,STEP *)
    IF xIN_Start THEN //IF rtSTART.Q THEN
        iOUT_Step := ST150_Uss_e.START;
    END_IF

(***** START  ZYKLISCH *****)
ST150_Uss_e.START: (*  *)
    IF xIN_NextStep AND pxFG_Freigabe^ THEN
        iOUT_Step := ST150_Uss_e.waitOnMover;
        iPreStep  := ST150_Uss_e.INIT;
    END_IF;

ST150_Uss_e.waitOnMover: (*  *)
    IF xIN_NextStep AND __ISVALIDREF(Mover) THEN
        IF Mover.GetLastStationDone() >= iIN_StationNumber THEN
            iOUT_Step := ST150_Uss_e.SYNC_MOVER_LEAVE;
        ELSIF Mover.GetLastStationDone() < INT#145 THEN
            iOUT_Step := ST150_Uss_e.SYNC_MOVER_LEAVE;
        ELSE
            iOUT_Step := ST150_Uss_e.check_cap_present;
            iPreStep  := ST150_Uss_e.waitOnMover;
        END_IF
    END_IF;

ST150_Uss_e.check_cap_present:
    IF xIN_capDetector OR (USS_SIMULATION AND CONST.USE_SIMULATION) THEN
        iOUT_Step := ST150_Uss_e.mover_maintening_up;
    ELSIF TON_CapDetection.Q THEN
        // Mover.SetErrorCode(CONCAT(CONCAT(INT_TO_STRING(iIN_StationNumber), '-B '), sIN_errorCodeSide));
        bOUT_Error := 8; // TODO to be removed
    END_IF

ST150_Uss_e.mover_maintening_up:
    IF xIN_NextStep AND fb_moverMaintening.xOUT_inAS THEN
        IF USS_SIMULATION AND CONST.USE_SIMULATION THEN
            iOUT_Step := ST150_Uss_e.mover_maintening_down;
        ELSE
            IF xIN_welding_bits.Bereit THEN
                iOUT_Step := ST150_Uss_e.uss_start;
                iPreStep  := ST150_Uss_e.waitOnMover;

                IF __ISVALIDREF(Mover) THEN
                    IF NOT Mover.SetLastStation(iIN_StationNumber) THEN
                        ASSERT(0);
                    END_IF
                END_IF
            ELSE
                // bOUT_Error := 1; // welding not ready
            END_IF
        END_IF;
    END_IF;

ST150_Uss_e.uss_start:
    IF xIN_NextStep AND NOT xIN_welding_bits.NullPosition THEN
        iOUT_Step := ST150_Uss_e.uss_working;
    END_IF

ST150_Uss_e.uss_working:
    IF xIN_NextStep AND
       (NOT xIN_welding_bits.US_on AND
       xIN_welding_bits.NullPosition) THEN
        iOUT_Step := ST150_Uss_e.mover_maintening_down;
    END_IF

ST150_Uss_e.mover_maintening_down:
    IF xIN_NextStep AND fb_moverMaintening.xOUT_inGS THEN
        iOUT_Step := ST150_Uss_e.SYNC_MOVER_LEAVE;

        IF __ISVALIDREF(Mover) THEN
            IF NOT Mover.SetLastStation(iIN_StationNumber) THEN
                ASSERT(0);
            END_IF
        END_IF
    END_IF;

ST150_Uss_e.SYNC_MOVER_LEAVE:
    // The mover needs to be taken by MoverMan
    IF NOT __ISVALIDREF(Mover) THEN
        iOUT_Step := ST150_Uss_e.DONE;
    END_IF

(***** DONE *****)
ST150_Uss_e.DONE: (* Letzter Schritt  *)
    IF NOT xIN_AlarmAktiv THEN
        //AUTO
        IF (enIN_State = StateAUTO) AND xIN_RestartCYCL THEN
            iOUT_Step := ST150_Uss_e.START;
            //STEP / END / LEERFAHREN restart
        ELSIF (enIN_State < StateAUTO) AND (enIN_State >= enState.StateSTEP) AND xIN_RestartCYCL THEN
            iOUT_Step := ST150_Uss_e.START;
            //STEP / END / LEERFAHREN fertig
        ELSIF (enIN_State = StateREADY) THEN
            iOUT_Step := ST150_Uss_e.READY;
        END_IF;
    END_IF;

(************ ERROR *************)
ST150_Uss_e.ERROR: (* ERROR *) ;

END_CASE;

END_FUNCTION_BLOCK

// ---- POUs/20_AUTO/ST15x/FB_AUT_155.TcPOU
FUNCTION_BLOCK FB_AUT_155 EXTENDS FB_AUT_ABSTRACT
(****************************************************************************)
(*	POU_AUT_zxx			Bausteinaufrufe Station	zxx							*)
(*	Status				ungetestet											*)
(*  Version:			1.0													*)
(*	Beschrieb:																*)
(*																			*)
(*	Abläufe:			FB_ABLzxxA		Hauptablauf							*)
(*																			*)
(*																			*)
(* 	25.09.2019/Dj															*)
(****************************************************************************)
(*	dd.mm.yyyy   KZ    x.y			Beschrieb								*)
(****************************************************************************)
VAR_INPUT
    (* spezifische Eingänge *)

END_VAR
VAR_OUTPUT
    (* spezifische Ausgänge *)

END_VAR
VAR
    (* Bausteine *)
    fb_Uss : FB_ABL_150;

    fb_stat : FB_AUT_Statistics;

END_VAR

(*******************************************************************)
(* Timer *)
(*******************************************************************)

(*******************************************************************)
(* Flanken / Merker *)
(*******************************************************************)
//MANU CYCLE
IF (enIN_State = StateMANU) AND xIN_ManuCycle THEN
    xManuCycle := TRUE;
END_IF;

IF (enIN_State <> StateMANU) OR xOUT_Done THEN
    xManuCycle := FALSE;
END_IF

//NEXT STEP
xNextStep := (enIN_State > StateSTEP) OR
             ((enIN_State = StateSTEP) AND xIN_Step) OR
             ((enIN_State = StateMANU) AND xManuCycle);

//RESET
xReset := (enIN_State < StateREADY) AND (enIN_State <> StateINIT) AND NOT xManuCycle;

(*******************************************************************)
(* Bausteinaufrufe Abläufe *)
(*******************************************************************)

xRelease := MAIN.MoverMan.IsProcessUsed(THIS^);

fb_Uss.xIN_welding_bits.Bereit       := IN.I024_ultraschall_bereit_155_20;
fb_Uss.xIN_welding_bits.Fehler       := IN.I025_ultraschall_fehler_155_20;
fb_Uss.xIN_welding_bits.US_on        := IN.I026_ultraschall_us_on_155_20;
fb_Uss.xIN_welding_bits.NullPosition := IN.I027_ultraschall_nullpos_155_20;

fb_Uss(xIN_Reset       := xReset,
       xIN_Init        := xIN_Init,
       xIN_Quit        := xIN_Quit,
       xIN_Start       := enIN_State >= enState.StateLEER AND xRelease,
       xIN_Sperre      := NOT xIN_On,
       xIN_NextStep    := xNextStep,
       xIN_AlarmAktiv  := xIN_AlarmAktiv,
       xIN_DryCycle    := xIN_DryCycle,
       xIN_RestartCYCL := enIN_State >= enState.StateLEER,
       enIN_State      := enIN_State,
       tIN_Timeout     := tIN_Timeout,
       pxFG_Freigabe   := ADR(xRelease),
       // CleverTrackLib
       Mover := THIS^.Mover,
       // hardware input
       xIN_capDetector             := IO_BOX.I2306_ST155_deckel_vohanden,
       xIN_kraftubersetzunh_zuruck := IO_BOX.I2304_ST155_kraftubersetzung_zuruck,
       xIN_kraftubersetzunh_vor    := IO_BOX.I2305_ST155_kraftubersetzung_vor,
       pIN_ButtonMaintaining       := ADR(HMI.btManuCylinders[StationList_e.ST155][1]),
       xIN_welding_bits            :=, // set above
       iIN_StationNumber           := 155,
       sIN_errorCodeSide           := 'Right',
       // hardware output
       xOUT_moverMaintening_valve => IO_BOX.Q0203_14_ST155_kraftubersetzung,
       xOUT_welding_bits          =>); // set below

OUT.Q030_ST155_ultraschall_start      := fb_Uss.xOUT_welding_bits.Start;
OUT.Q031_ST155_ultraschall_reset      := fb_Uss.xOUT_welding_bits.Reset;
OUT.Q032_ST155_ultraschall_data_bit_0 := fb_Uss.xOUT_welding_bits.Data_Hex1;
OUT.Q033_ST155_ultraschall_data_bit_1 := fb_Uss.xOUT_welding_bits.Data_Hex2;
OUT.Q034_ST155_ultraschall_data_bit_2 := fb_Uss.xOUT_welding_bits.Data_Hex4;
OUT.Q035_ST155_ultraschall_data_bit_3 := fb_Uss.xOUT_welding_bits.Data_Hex8;

fb_stat(xIN_Enable  := enState.StateAUTO = enIN_State,
        xIN_Waiting := fb_Uss.xOUT_Wait,
        xIN_Running := (fb_Uss.iOUT_Step >= ST150_Uss_e.START) AND
                       (fb_Uss.iOUT_Step <= ST150_Uss_e.DONE),
        // Since we use a mover system, a cycle is done when we are waiting on a mover
        xIN_Done := fb_Uss.iOUT_Step = ST150_Uss_e.waitOnMover);

(*******************************************************************)
(* Mover reset flags *)
(*******************************************************************)

(*******************************************************************)
(* OUTPUT *)
(*******************************************************************)
xOUT_InitDone := fb_Uss.xOUT_InitDone;
xOUT_Ready    := fb_Uss.xOUT_Ready;
xOUT_Done     := fb_Uss.xOUT_Done;
xOUT_ErrFlag  := fb_Uss.xOUT_ErrFlag;
xOUT_Wait     := fb_Uss.xOUT_Wait;
xOUT_AlarmST  := xOUT_ErrFlag;

(*******************************************************************)
(* Bausteinaufruf Error Station *)
(*******************************************************************)
// POU_ERR_VORLAGE(xIN_QUIT:=xIN_Quit , pstrArIN_ALARM:=ADR(HMI.strArALARM[1]));

(* % of completion of the process *)
PROPERTY iCompletionPC : INT
GET
iCompletionPC := THIS^.fb_Uss.iOUT_ProcessCompletion;
END_GET
END_PROPERTY

PROPERTY ProcessExecution : ProcessExecution_e
GET
ProcessExecution := THIS^._ProcessExecution;
END_GET
SET
THIS^._ProcessExecution := ProcessExecution;
END_SET
END_PROPERTY

PROPERTY xBusy : BOOL
GET
xBusy := THIS^.fb_Uss.xOUT_Busy;
END_GET
SET
END_SET
END_PROPERTY

PROPERTY xDone : BOOL
GET
xDone := THIS^.fb_Uss.xOUT_Ready OR THIS^.fb_Uss.xOUT_Done;
END_GET
END_PROPERTY

PROPERTY xMoverPathFree : BOOL
GET
xMoverPathFree := THIS^.fb_Uss.xOUT_MoverFree OR THIS^.fb_Uss.xOUT_Ready OR THIS^.fb_Uss.xOUT_Done;
END_GET
END_PROPERTY

PROPERTY xMoverShouldLeave : BOOL
GET
xMoverShouldLeave := THIS^.fb_Uss.iOUT_Step = ST150_Uss_e.SYNC_MOVER_LEAVE;
END_GET
END_PROPERTY

END_FUNCTION_BLOCK

// ---- POUs/20_AUTO/ST16x/FB_AUT_160.TcPOU
FUNCTION_BLOCK FB_AUT_160 EXTENDS FB_AUT_ABSTRACT
(****************************************************************************)
(*	POU_AUT_zxx			Bausteinaufrufe Station	zxx							*)
(*	Status				ungetestet											*)
(*  Version:			1.0													*)
(*	Beschrieb:																*)
(*																			*)
(*	Abläufe:			FB_ABLzxxA		Hauptablauf							*)
(*																			*)
(*																			*)
(* 	25.09.2019/Dj															*)
(****************************************************************************)
(*	dd.mm.yyyy   KZ    x.y			Beschrieb								*)
(****************************************************************************)
VAR_INPUT
    (* spezifische Eingänge *)

END_VAR
VAR_OUTPUT
    (* spezifische Ausgänge *)

END_VAR
VAR
    (* Bausteine *)
    fb_ABL_CETA : FB_ABL_160;
	
	ceta_160 : FB_CETA_715;

    fb_stat : FB_AUT_Statistics;

END_VAR

(*******************************************************************)
(* Timer *)
(*******************************************************************)

(*******************************************************************)
(* Flanken / Merker *)
(*******************************************************************)
//MANU CYCLE
IF (enIN_State = StateMANU) AND xIN_ManuCycle THEN
    xManuCycle := TRUE;
END_IF;

IF (enIN_State <> StateMANU) OR xOUT_Done THEN
    xManuCycle := FALSE;
END_IF

//NEXT STEP
xNextStep := (enIN_State > StateSTEP) OR
             ((enIN_State = StateSTEP) AND xIN_Step) OR
             ((enIN_State = StateMANU) AND xManuCycle);

//RESET
xReset := (enIN_State < StateREADY) AND (enIN_State <> StateINIT) AND NOT xManuCycle;

(*******************************************************************)
(* Bausteinaufrufe Abläufe *)
(*******************************************************************)

xRelease := MAIN.MoverMan.IsProcessUsed(THIS^);

ceta_160(xIN_StatusBits   := CETA_IO.I_ST160_StatusBits,
         xIN_Data         := CETA_IO.I_ST160_Data,
         xIN_Reset        := xReset OR xIN_Quit,
         xOUT_CommandBits => CETA_IO.Q_ST160_CommandBits,
         xOUT_Data        => CETA_IO.Q_ST160_Data);

fb_ABL_CETA(xIN_Reset       := xReset,
            xIN_Init        := xIN_Init,
            xIN_Quit        := xIN_Quit,
            xIN_Start       := enIN_State >= enState.StateLEER AND xRelease,
            xIN_Sperre      := NOT xIN_On,
            xIN_NextStep    := xNextStep,
            xIN_AlarmAktiv  := xIN_AlarmAktiv,
            xIN_DryCycle    := xIN_DryCycle,
            xIN_RestartCYCL := enIN_State >= enState.StateLEER,
            enIN_State      := enIN_State,
            tIN_Timeout     := tIN_Timeout,
            pxFG_Freigabe   := ADR(xRelease),
            // CleverTrackLib
            Mover := THIS^.Mover,
            // for multiple reference of the FB
            ref_fb_CETA := ceta_160,

            refAxis_01Z_beckhoff         := ST16x_Axis.axis160_01Z,
            constAxis_01Z_Beckhoff       := ST16x_Axis.const160_01Z,
            axis_01Z_LinearConfig        := _20_AUTO.recipe.linearAxis[LinearAxis_e.ST160_01Z],
            iSelectedAxis                := Axis_e.ST160_01Z,
            axis_01Z_parIN_Buttons       := ADR(AXIS.btTeachArAxis[Axis_e.ST160_01Z]),
            refCylinderBp                := HMI.btManuCylinders[StationList_e.ST160],
            refCylinderConf              := _20_AUTO.recipe.cylinder2Pos[StationList_e.ST160],
            uiIN_DisplacementSensorLeft  := IO_BOX.I3000_ST160_Wegmessenor_links,
            uiIN_DisplacementSensorRight := IO_BOX.I3100_ST160_Wegmessenor_rechts,
            IN_recipe                    := _20_AUTO.recipe.st160,
            iIN_StationNumber            := 160,

            xOUT_niederhalter_links         => IO_BOX.Q0300_14_ST160_niederhalter_links,
            xOUT_niederhalter_rechts        => IO_BOX.Q0301_14_ST160_niederhalter_rechts,
            xOUT_dichtung_pruflocker_links  => IO_BOX.Q0302_14_ST160_dichtung_pruflocker_links,
            xOUT_dichtung_pruflocker_rechts => IO_BOX.Q0302_12_ST160_dichtung_pruflocker_rechts,

            axisRef_Hardware   := ST16x_Axis.axis160_01Z.axis,
            axisRef_Simulation := SIMU.axis_ref[Axis_e.ST160_01Z]);

fb_stat(xIN_Enable  := enState.StateAUTO = enIN_State,
        xIN_Waiting := fb_ABL_CETA.xOUT_Wait,
        xIN_Running := (fb_ABL_CETA.iOUT_Step >= ST160_CETA_e.START) AND
                       (fb_ABL_CETA.iOUT_Step <= ST160_CETA_e.DONE),
        // Since we use a mover system, a cycle is done when we are waiting on a mover
        xIN_Done := fb_ABL_CETA.iOUT_Step = ST160_CETA_e.waitOnMover);

(*******************************************************************)
(* Mover reset flags *)
(*******************************************************************)

(*******************************************************************)
(* OUTPUT *)
(*******************************************************************)
xOUT_InitDone := fb_ABL_CETA.xOUT_InitDone;
xOUT_Ready    := fb_ABL_CETA.xOUT_Ready;
xOUT_Done     := fb_ABL_CETA.xOUT_Done;
xOUT_ErrFlag  := fb_ABL_CETA.xOUT_ErrFlag;
xOUT_Wait     := fb_ABL_CETA.xOUT_Wait;
xOUT_AlarmST  := xOUT_ErrFlag;

(*******************************************************************)
(* Bausteinaufruf Error Station *)
(*******************************************************************)
// POU_ERR_VORLAGE(xIN_QUIT:=xIN_Quit , pstrArIN_ALARM:=ADR(HMI.strArALARM[1]));

(* % of completion of the process *)
PROPERTY iCompletionPC : INT
GET
iCompletionPC := THIS^.fb_ABL_CETA.iOUT_ProcessCompletion;
END_GET
END_PROPERTY

PROPERTY ProcessExecution : ProcessExecution_e
GET
ProcessExecution := THIS^._ProcessExecution;
END_GET
SET
THIS^._ProcessExecution := ProcessExecution;
END_SET
END_PROPERTY

PROPERTY xBusy : BOOL
GET
xBusy := THIS^.fb_ABL_CETA.xOUT_Busy;
END_GET
SET
END_SET
END_PROPERTY

PROPERTY xDone : BOOL
GET
xDone := THIS^.fb_ABL_CETA.xOUT_Ready OR THIS^.fb_ABL_CETA.xOUT_Done;
END_GET
END_PROPERTY

PROPERTY xMoverPathFree : BOOL
GET
xMoverPathFree := THIS^.fb_ABL_CETA.xOUT_MoverFree OR THIS^.fb_ABL_CETA.xOUT_Ready OR THIS^.fb_ABL_CETA.xOUT_Done;
END_GET
END_PROPERTY

PROPERTY xMoverShouldLeave : BOOL
GET
xMoverShouldLeave := THIS^.fb_ABL_CETA.iOUT_Step = ST160_CETA_e.SYNC_MOVER_LEAVE;
END_GET
END_PROPERTY

END_FUNCTION_BLOCK

// ---- POUs/20_AUTO/ST16x/FB_ABL_160.TcPOU
FUNCTION_BLOCK FB_ABL_160
(****************************************************************************************)
(*	TITEL				laden kristall- Modul	    										*)
(*	Status				ungetestet                         								*)
(*	Beschrieb:			Ablaufbeschreibung												*)
(*																						*)
(*	Steps:	self-explained using enum													*)
(***********************************Revisionen*******************************************)
(*	see github blames																	*)
(****************************************************************************************)

VAR_INPUT
    xIN_Reset       : BOOL;          // Schrittkette zurücksetzen 
    xIN_Init        : BOOL;          // Initialisieren
    xIN_Quit        : BOOL;          // Fehler quittieren 
    xIN_Start       : BOOL;          // Startbefehl
    xIN_Sperre      : BOOL;          // FB Sperren 
    xIN_NextStep    : BOOL;          // Nächsten Schritt ausführen 
    xIN_AlarmAktiv  : BOOL;          // Anlage hat Alarm
    xIN_DryCycle    : BOOL;          // Fahren ohne Teile
    xIN_RestartCYCL : BOOL;          // Zyklus erneut starten im STEP, END, LEERFAHREN
    enIN_State      : enState;       // Status Anlage
    tIN_Timeout     : TIME := T#10s; // Timout

    pxFG_Freigabe : POINTER TO BOOL; //Freigabe von Station

    // Application specific
    Mover                  : REFERENCE TO FB_Mover;
    ref_fb_CETA            : REFERENCE TO FB_CETA_715;
    refAxis_01Z_beckhoff   : REFERENCE TO AxisBeckhoff_t; // reference of the axis GVL struct
    constAxis_01Z_Beckhoff : AxisLinMotConst_t;
    axis_01Z_LinearConfig  : LinearMotionMan_Config_t;
    iSelectedAxis          : Axis_e;
    axis_01Z_parIN_Buttons : POINTER TO ARRAY[0..8] OF structButton;
    refCylinderBp          : REFERENCE TO ARRAY[0..CONST.MAX_CYLINDER_PER_STATION] OF structButton;
    refCylinderConf        : REFERENCE TO ARRAY[0..CONST.MAX_CYLINDER_PER_STATION] OF Cylinder2Pos_config;

    // inputs
    uiIN_DisplacementSensorLeft  : UINT;
    uiIN_DisplacementSensorRight : UINT;
    IN_recipe                    : ST160_Recipe_t;
    iIN_StationNumber            : INT;

END_VAR
VAR_OUTPUT
    (* standart Ausgänge *)
    xOUT_ErrFlag  : BOOL;         // Error Flag 
    xOUT_Busy     : BOOL;         // Baustein befindet sich im Ablauf 
    xOUT_Done     : BOOL;         // Baustein hat den Ablauf beendet 		
    xOUT_Ready    : BOOL;         // Ready to begin, should be the same state as done	
    xOUT_Timeout  : BOOL;         // Timeout FB 
    xOUT_InitDone : BOOL;         // initialisierung fertig
    xOUT_Wait     : BOOL;         // Wartet auf Bedingung
    iOUT_Step     : ST160_CETA_e; // Aktueller Schritt 
    sOUT_Step     : STRING;       // Aktueller Schritt but in string format
    bOUT_Error    : BYTE;         // Fehlernummer

    iOUT_ProcessCompletion : INT;  //process completion, express in % (0-100)
    xOUT_MoverFree         : BOOL; // The mover is free to move

    // outputs
    xOUT_niederhalter_links         : BOOL;
    xOUT_niederhalter_rechts        : BOOL;
    xOUT_dichtung_pruflocker_links  : BOOL;
    xOUT_dichtung_pruflocker_rechts : BOOL;

END_VAR
VAR
    (* Standard *)
    (* Schritt *)
    iLastStep : ST160_CETA_e; // Merker letzter Schritt 
    iPreStep  : ST160_CETA_e; // Schritt zurück nach Alarm 
    iAktStep  : ST160_CETA_e; // aktueller Schritt

    // Trigger Starten 
    rtSTART : R_TRIG;
    // Timer TimeOut 
    TON_Timeout : TON;

    (* Bausteine *)
    fb_PnpVerAxis    : FB_LinearMotionMan;
    simu_axis160_01Z : FB_Simu_AxisLIN_V1_1;
    fb_axis160_01Z   : FB_AxisLIN_V1_1;

    (* Spezial *)
    fb_capMainteningLeft  : FB_ZylMo2El_V2_1;
    fb_capMainteningRight : FB_ZylMo2El_V2_1;

    simu_capMainteningLeft  : FB_Simu_Zyl2Pos;
    simu_capMainteningRight : FB_Simu_Zyl2Pos;

    fb_dichtung_left  : FB_ZylMo2El_V2_1;
    fb_dichtung_right : FB_ZylMo2El_V2_1;

    simu_dichtung_left  : FB_Simu_Zyl2Pos;
    simu_dichtung_right : FB_Simu_Zyl2Pos;

    xCETA_Result_OK : BOOL;
END_VAR

VAR_IN_OUT
    axisRef_Hardware   : AXIS_REF;
    axisRef_Simulation : AXIS_REF;
END_VAR

VAR CONSTANT
    CETA_SIMULATION : BOOL := FALSE; // Set to TRUE to simulate this part of the program
END_VAR

